C05463=1086.064,-73.363,-52.991,174.293,17.669,152.886
C05464=1086.058,-73.613,-52.980,174.292,17.667,152.886
C05465=1086.052,-73.862,-52.969,174.290,17.666,152.886
C05466=1086.046,-74.112,-52.958,174.289,17.665,152.886
C05467=1086.040,-74.362,-52.947,174.287,17.664,152.887
C05468=1086.034,-74.611,-52.936,174.286,17.662,152.886
C05469=1086.028,-74.861,-52.925,174.284,17.661,152.887
C05470=1086.021,-75.111,-52.914,174.282,17.660,152.887
C05471=1086.016,-75.360,-52.903,174.281,17.658,152.887
C05472=1086.010,-75.610,-52.892,174.279,17.657,152.887
C05473=1086.004,-75.860,-52.881,174.278,17.656,152.887
C05474=1085.998,-76.110,-52.870,174.277,17.655,152.887
C05475=1085.992,-76.359,-52.859,174.275,17.654,152.887
C05476=1085.986,-76.608,-52.849,174.274,17.653,152.887
C05477=1085.979,-76.858,-52.838,174.272,17.652,152.887
C05478=1085.974,-77.108,-52.827,174.271,17.650,152.887
C05479=1085.968,-77.358,-52.817,174.269,17.649,152.887
C05480=1085.962,-77.607,-52.806,174.268,17.648,152.887
C05481=1085.956,-77.858,-52.795,174.266,17.646,152.887
C05482=1085.950,-78.107,-52.785,174.265,17.645,152.887
C05483=1085.944,-78.356,-52.774,174.263,17.644,152.887
C05484=1085.938,-78.607,-52.762,174.261,17.643,152.887
C05485=1085.932,-78.856,-52.752,174.260,17.642,152.887
C05486=1085.926,-79.105,-52.741,174.258,17.640,152.887
C05487=1085.921,-79.356,-52.730,174.257,17.639,152.887
C05488=1085.914,-79.605,-52.720,174.255,17.638,152.888
C05489=1085.908,-79.855,-52.709,174.254,17.636,152.888
C05490=1085.902,-80.104,-52.698,174.252,17.635,152.888
C05491=1085.896,-80.354,-52.687,174.250,17.634,152.888
C05492=1085.889,-80.604,-52.677,174.250,17.634,152.888
C05493=1085.883,-80.879,-52.665,174.247,17.631,152.888
C05494=1085.876,-81.154,-52.654,174.246,17.630,152.888
C05495=1085.870,-81.429,-52.642,174.244,17.629,152.888
C05496=1085.863,-81.705,-52.629,174.243,17.628,152.888
C05497=1085.857,-81.955,-52.619,174.241,17.627,152.888
C05498=1085.851,-82.204,-52.609,174.239,17.626,152.888
C05499=1085.845,-82.454,-52.598,174.238,17.625,152.888
C05500=1085.839,-82.704,-52.587,174.236,17.623,152.888
C05501=1085.832,-82.953,-52.577,174.235,17.622,152.888
C05502=1085.827,-83.203,-52.566,174.233,17.621,152.889
C05503=1085.820,-83.452,-52.556,174.232,17.620,152.889
C05504=1085.814,-83.703,-52.545,174.231,17.619,152.889
C05505=1085.808,-83.952,-52.534,174.229,17.618,152.889
C05506=1085.802,-84.202,-52.524,174.227,17.617,152.889
C05507=1085.796,-84.451,-52.514,174.226,17.616,152.889
C05508=1085.790,-84.702,-52.502,174.224,17.615,152.889
C05509=1085.784,-84.951,-52.493,174.223,17.613,152.889
C05510=1085.778,-85.201,-52.482,174.221,17.612,152.889
C05511=1085.771,-85.450,-52.472,174.219,17.611,152.889
C05512=1085.766,-85.699,-52.461,174.218,17.610,152.889
C05513=1085.760,-85.950,-52.450,174.216,17.608,152.889
C05514=1085.753,-86.199,-52.440,174.216,17.608,152.889
C05515=1085.747,-86.449,-52.429,174.214,17.607,152.889
C05516=1085.741,-86.699,-52.419,174.212,17.606,152.890
C05517=1085.736,-86.948,-52.409,174.211,17.604,152.890
C05518=1085.729,-87.198,-52.397,174.209,17.603,152.890
C05519=1085.723,-87.448,-52.388,174.208,17.602,152.890
C05520=1085.717,-87.698,-52.377,174.206,17.601,152.890
C05521=1085.711,-87.947,-52.367,174.204,17.600,152.890
C05522=1085.705,-88.197,-52.356,174.203,17.599,152.890
C05523=1085.699,-88.446,-52.346,174.201,17.597,152.890
C05524=1085.693,-88.697,-52.336,174.200,17.596,152.890
C05525=1085.687,-88.947,-52.325,174.199,17.595,152.890
C05526=1085.681,-89.196,-52.314,174.197,17.594,152.890
C05527=1085.675,-89.446,-52.304,174.195,17.593,152.890
C05528=1085.669,-89.695,-52.294,174.194,17.592,152.891
C05529=1085.663,-89.945,-52.284,174.192,17.591,152.891
C05530=1085.656,-90.195,-52.273,174.191,17.590,152.891
C05531=1085.650,-90.444,-52.262,174.189,17.589,152.891
C05532=1085.645,-90.695,-52.252,174.187,17.587,152.891
C05533=1085.639,-90.944,-52.242,174.187,17.587,152.891
C05534=1085.633,-91.194,-52.232,174.185,17.586,152.891
C05535=1085.627,-91.443,-52.221,174.183,17.585,152.891
C05536=1085.621,-91.693,-52.211,174.182,17.583,152.891
C05537=1085.615,-91.942,-52.201,174.180,17.582,152.891
C05538=1085.609,-92.193,-52.190,174.179,17.581,152.891
C05539=1085.602,-92.442,-52.180,174.177,17.580,152.891
C05540=1085.597,-92.692,-52.170,174.175,17.579,152.892
C05541=1085.590,-92.942,-52.160,174.174,17.578,152.892
C05542=1085.585,-93.192,-52.150,174.173,17.577,152.892
C05543=1085.578,-93.441,-52.139,174.171,17.576,152.892
C05544=1085.573,-93.691,-52.129,174.170,17.575,152.892
C05545=1085.567,-93.940,-52.119,174.168,17.574,152.892
C05546=1085.561,-94.190,-52.109,174.166,17.573,152.892
C05547=1085.555,-94.439,-52.098,174.165,17.572,152.892
C05548=1085.549,-94.690,-52.088,174.163,17.570,152.892
C05549=1085.543,-94.939,-52.078,174.162,17.570,152.892
C05550=1085.537,-95.189,-52.068,174.161,17.569,152.892
C05551=1085.530,-95.439,-52.057,174.159,17.568,152.893
C05552=1085.525,-95.689,-52.047,174.157,17.567,152.893
C05553=1085.518,-95.938,-52.037,174.156,17.566,152.893
C05554=1085.513,-96.188,-52.027,174.154,17.564,152.893
C05555=1085.507,-96.438,-52.017,174.153,17.563,152.893
C05556=1085.501,-96.687,-52.006,174.152,17.563,152.893
C05557=1085.494,-96.964,-51.995,174.150,17.561,152.893
C05558=1085.488,-97.242,-51.984,174.148,17.560,152.893
C05559=1085.481,-97.520,-51.972,174.146,17.559,152.893
C05560=1085.474,-97.797,-51.962,174.144,17.558,152.893
C05561=1085.469,-98.047,-51.951,174.144,17.557,152.894
C05562=1085.462,-98.297,-51.941,174.142,17.556,152.894
C05563=1085.455,-98.547,-51.931,174.140,17.555,152.894
C05564=1085.450,-98.797,-51.921,174.139,17.554,152.894
C05565=1085.444,-99.046,-51.911,174.137,17.553,152.894
C05566=1085.437,-99.296,-51.901,174.135,17.552,152.894
C05567=1085.432,-99.546,-51.891,174.134,17.551,152.894
C05568=1085.425,-99.795,-51.881,174.133,17.550,152.894
C05569=1085.419,-100.045,-51.871,174.131,17.549,152.894
C05570=1085.414,-100.295,-51.861,174.129,17.548,152.894
C05571=1085.407,-100.544,-51.851,174.128,17.547,152.895
C05572=1085.401,-100.794,-51.841,174.126,17.546,152.895
C05573=1085.395,-101.044,-51.832,174.125,17.546,152.895
C05574=1085.389,-101.293,-51.821,174.123,17.545,152.895
C05575=1085.383,-101.543,-51.811,174.122,17.544,152.895
C05576=1085.377,-101.793,-51.802,174.120,17.543,152.895
C05577=1085.371,-102.043,-51.792,174.118,17.542,152.895
C05578=1085.365,-102.292,-51.781,174.117,17.541,152.895
C05579=1085.359,-102.542,-51.772,174.116,17.540,152.896
C05580=1085.353,-102.792,-51.762,174.114,17.539,152.896
C05581=1085.347,-103.041,-51.751,174.113,17.538,152.896
C05582=1085.341,-103.291,-51.742,174.111,17.537,152.896
C05583=1085.335,-103.541,-51.732,174.109,17.536,152.896
C05584=1085.328,-103.791,-51.722,174.108,17.535,152.896
C05585=1085.323,-104.041,-51.712,174.107,17.535,152.896
C05586=1085.317,-104.290,-51.702,174.105,17.534,152.896
C05587=1085.310,-104.540,-51.692,174.103,17.533,152.897
C05588=1085.304,-104.789,-51.683,174.102,17.532,152.897
C05589=1085.298,-105.039,-51.673,174.100,17.531,152.897
C05590=1085.292,-105.289,-51.662,174.099,17.530,152.897
C05591=1085.286,-105.538,-51.653,174.097,17.529,152.897
C05592=1085.280,-105.788,-51.643,174.096,17.528,152.897
C05593=1085.274,-106.038,-51.634,174.094,17.527,152.897
C05594=1085.268,-106.288,-51.624,174.092,17.526,152.897
C05595=1085.262,-106.537,-51.613,174.091,17.526,152.898
C05596=1085.256,-106.787,-51.604,174.090,17.525,152.898
C05597=1085.250,-107.037,-51.594,174.088,17.524,152.898
C05598=1085.243,-107.287,-51.585,174.086,17.523,152.898
C05599=1085.237,-107.537,-51.575,174.084,17.522,152.898
C05600=1085.232,-107.787,-51.565,174.084,17.522,152.898
C05601=1085.226,-108.036,-51.555,174.082,17.521,152.898
C05602=1085.219,-108.286,-51.545,174.080,17.519,152.898
C05603=1085.213,-108.535,-51.535,174.079,17.518,152.899
C05604=1085.207,-108.785,-51.526,174.078,17.518,152.899
C05605=1085.201,-109.035,-51.516,174.076,17.517,152.899
C05606=1085.194,-109.285,-51.507,174.074,17.516,152.899
C05607=1085.188,-109.535,-51.497,174.073,17.515,152.899
C05608=1085.182,-109.784,-51.488,174.071,17.515,152.899
C05609=1085.176,-110.034,-51.478,174.070,17.514,152.899
C05610=1085.169,-110.283,-51.468,174.068,17.513,152.900
C05611=1085.164,-110.534,-51.458,174.067,17.512,152.900
C05612=1085.158,-110.783,-51.448,174.065,17.511,152.900
C05613=1085.152,-111.033,-51.438,174.064,17.511,152.900
C05614=1085.145,-111.283,-51.429,174.062,17.510,152.900
C05615=1085.139,-111.533,-51.419,174.060,17.509,152.900
C05616=1085.133,-111.783,-51.410,174.059,17.508,152.900
C05617=1085.128,-112.032,-51.400,174.057,17.507,152.901
C05618=1085.121,-112.281,-51.391,174.056,17.507,152.901
C05619=1085.115,-112.531,-51.381,174.054,17.506,152.901
C05620=1085.109,-112.781,-51.372,174.052,17.505,152.901
C05621=1085.103,-113.054,-51.361,174.051,17.504,152.901
C05622=1085.095,-113.327,-51.350,174.049,17.503,152.901
C05623=1085.089,-113.600,-51.340,174.047,17.502,152.902
C05624=1085.082,-113.873,-51.330,174.046,17.501,152.902
C05625=1085.076,-114.123,-51.320,174.045,17.501,152.902
C05626=1085.070,-114.373,-51.311,174.043,17.500,152.902
C05627=1085.064,-114.622,-51.301,174.041,17.499,152.902
C05628=1085.058,-114.872,-51.292,174.040,17.498,152.902
C05629=1085.052,-115.122,-51.282,174.038,17.498,152.902
C05630=1085.046,-115.371,-51.273,174.037,17.497,152.903
C05631=1085.040,-115.621,-51.263,174.035,17.497,152.903
C05632=1085.033,-115.871,-51.254,174.033,17.495,152.903
C05633=1085.027,-116.121,-51.244,174.032,17.495,152.903
C05634=1085.021,-116.371,-51.234,174.030,17.494,152.903
C05635=1085.015,-116.620,-51.225,174.029,17.493,152.903
C05636=1085.009,-116.870,-51.215,174.027,17.492,152.903
C05637=1085.003,-117.120,-51.207,174.026,17.492,152.904
C05638=1084.997,-117.370,-51.197,174.024,17.491,152.904
C05639=1084.990,-117.619,-51.188,174.022,17.491,152.904
C05640=1084.984,-117.869,-51.179,174.022,17.490,152.904
C05641=1084.978,-118.119,-51.169,174.020,17.489,152.904
C05642=1084.972,-118.369,-51.160,174.018,17.489,152.905
C05643=1084.966,-118.618,-51.150,174.016,17.487,152.905
C05644=1084.959,-118.868,-51.140,174.015,17.487,152.905
C05645=1084.954,-119.117,-51.131,174.014,17.486,152.905
C05646=1084.948,-119.367,-51.122,174.012,17.486,152.905
C05647=1084.942,-119.617,-51.113,174.010,17.485,152.905
C05648=1084.936,-119.867,-51.103,174.009,17.484,152.905
C05649=1084.929,-120.117,-51.094,174.007,17.484,152.906
C05650=1084.923,-120.367,-51.085,174.006,17.483,152.906
C05651=1084.916,-120.616,-51.075,174.004,17.483,152.906
C05652=1084.911,-120.865,-51.066,174.003,17.482,152.906
C05653=1084.905,-121.116,-51.057,174.001,17.481,152.906
C05654=1084.899,-121.366,-51.048,173.999,17.480,152.906
C05655=1084.893,-121.615,-51.038,173.998,17.480,152.907
C05656=1084.886,-121.865,-51.029,173.996,17.479,152.907
C05657=1084.880,-122.115,-51.019,173.995,17.478,152.907
C05658=1084.874,-122.364,-51.010,173.994,17.478,152.907
C05659=1084.868,-122.614,-51.001,173.992,17.477,152.907
C05660=1084.862,-122.864,-50.992,173.990,17.476,152.908
C05661=1084.856,-123.114,-50.982,173.988,17.476,152.908
C05662=1084.849,-123.363,-50.973,173.987,17.475,152.908
C05663=1084.843,-123.614,-50.964,173.985,17.475,152.908
C05664=1084.837,-123.863,-50.955,173.984,17.474,152.908
C05665=1084.831,-124.113,-50.946,173.983,17.474,152.908
C05666=1084.825,-124.362,-50.936,173.981,17.472,152.909
C05667=1084.819,-124.613,-50.927,173.979,17.472,152.909
C05668=1084.812,-124.862,-50.918,173.978,17.471,152.909
C05669=1084.807,-125.111,-50.909,173.976,17.471,152.909
C05670=1084.801,-125.361,-50.899,173.975,17.470,152.909
C05671=1084.794,-125.611,-50.891,173.973,17.469,152.910
C05672=1084.788,-125.861,-50.882,173.972,17.469,152.910
C05673=1084.782,-126.111,-50.872,173.970,17.468,152.910
C05674=1084.775,-126.361,-50.863,173.968,17.468,152.910
C05675=1084.769,-126.610,-50.855,173.967,17.467,152.910
C05676=1084.763,-126.860,-50.845,173.965,17.467,152.910
C05677=1084.757,-127.110,-50.835,173.963,17.466,152.911
C05678=1084.750,-127.360,-50.827,173.963,17.466,152.911
C05679=1084.744,-127.610,-50.818,173.961,17.465,152.911
C05680=1084.739,-127.859,-50.808,173.959,17.464,152.911
C05681=1084.733,-128.116,-50.799,173.958,17.464,152.911
C05682=1084.731,-128.373,-50.789,173.957,17.462,152.911
C05683=1084.733,-128.628,-50.776,173.956,17.459,152.911
C05684=1084.740,-128.881,-50.763,173.955,17.454,152.910
C05685=1084.338,-128.903,-50.895,173.912,17.569,152.940
C05686=1084.332,-128.650,-50.909,173.912,17.573,152.941
C05687=1084.328,-128.394,-50.921,173.912,17.577,152.941
C05688=1084.331,-128.138,-50.932,173.914,17.578,152.941
C05689=1084.335,-127.881,-50.941,173.915,17.579,152.941
C05690=1084.342,-127.632,-50.950,173.917,17.580,152.941
C05691=1084.348,-127.382,-50.960,173.918,17.580,152.941
C05692=1084.354,-127.132,-50.969,173.920,17.581,152.941
C05693=1084.361,-126.882,-50.978,173.922,17.582,152.941
C05694=1084.367,-126.633,-50.987,173.923,17.582,152.940
C05695=1084.373,-126.383,-50.996,173.925,17.583,152.940
C05696=1084.379,-126.133,-51.005,173.927,17.584,152.940
C05697=1084.386,-125.883,-51.014,173.928,17.584,152.940
C05698=1084.392,-125.633,-51.023,173.929,17.585,152.940
C05699=1084.397,-125.384,-51.032,173.931,17.585,152.939
C05700=1084.404,-125.134,-51.041,173.933,17.586,152.939
C05701=1084.410,-124.884,-51.051,173.934,17.586,152.939
C05702=1084.416,-124.634,-51.060,173.936,17.587,152.939
C05703=1084.422,-124.384,-51.069,173.938,17.588,152.939
C05704=1084.428,-124.135,-51.078,173.938,17.588,152.939
C05705=1084.435,-123.886,-51.087,173.940,17.589,152.938
C05706=1084.441,-123.635,-51.096,173.942,17.590,152.938
C05707=1084.447,-123.385,-51.106,173.944,17.590,152.938
C05708=1084.453,-123.136,-51.115,173.945,17.591,152.938
C05709=1084.459,-122.886,-51.125,173.947,17.592,152.938
C05710=1084.466,-122.637,-51.133,173.948,17.593,152.937
C05711=1084.471,-122.387,-51.142,173.949,17.593,152.937
C05712=1084.478,-122.137,-51.152,173.951,17.594,152.937
C05713=1084.484,-121.887,-51.161,173.953,17.594,152.937
C05714=1084.490,-121.637,-51.171,173.955,17.595,152.937
C05715=1084.496,-121.387,-51.181,173.956,17.595,152.937
C05716=1084.501,-121.138,-51.189,173.957,17.596,152.936
C05717=1084.508,-120.888,-51.198,173.959,17.597,152.936
C05718=1084.514,-120.638,-51.208,173.961,17.598,152.936
C05719=1084.521,-120.389,-51.217,173.962,17.598,152.936
C05720=1084.527,-120.139,-51.227,173.964,17.599,152.936
C05721=1084.533,-119.889,-51.236,173.965,17.600,152.936
C05722=1084.538,-119.639,-51.245,173.966,17.601,152.936
C05723=1084.544,-119.390,-51.254,173.968,17.601,152.935
C05724=1084.551,-119.140,-51.264,173.970,17.602,152.935
C05725=1084.557,-118.890,-51.273,173.972,17.603,152.935
C05726=1084.564,-118.640,-51.282,173.973,17.603,152.935
C05727=1084.570,-118.391,-51.292,173.975,17.604,152.935
C05728=1084.576,-118.141,-51.302,173.976,17.605,152.934
C05729=1084.582,-117.891,-51.311,173.978,17.606,152.934
C05730=1084.588,-117.642,-51.320,173.979,17.606,152.934
C05731=1084.594,-117.392,-51.329,173.981,17.607,152.934
C05732=1084.600,-117.142,-51.339,173.982,17.608,152.934
C05733=1084.606,-116.892,-51.348,173.984,17.608,152.934
C05734=1084.612,-116.642,-51.358,173.985,17.609,152.934
C05735=1084.618,-116.392,-51.368,173.987,17.610,152.933
C05736=1084.624,-116.143,-51.377,173.989,17.611,152.933
C05737=1084.631,-115.893,-51.387,173.990,17.612,152.933
C05738=1084.638,-115.643,-51.396,173.991,17.612,152.933
C05739=1084.643,-115.394,-51.405,173.993,17.613,152.933
C05740=1084.649,-115.144,-51.414,173.995,17.614,152.933
C05741=1084.655,-114.895,-51.424,173.996,17.615,152.932
C05742=1084.662,-114.645,-51.434,173.998,17.615,152.932
C05743=1084.668,-114.395,-51.443,173.999,17.616,152.932
C05744=1084.674,-114.145,-51.453,174.001,17.617,152.932
C05745=1084.680,-113.895,-51.462,174.003,17.617,152.932
C05746=1084.686,-113.622,-51.473,174.004,17.619,152.932
C05747=1084.693,-113.348,-51.484,174.005,17.619,152.932
C05748=1084.700,-113.075,-51.494,174.007,17.620,152.931
C05749=1084.706,-112.802,-51.504,174.009,17.621,152.931
C05750=1084.712,-112.552,-51.514,174.011,17.622,152.931
C05751=1084.718,-112.303,-51.523,174.012,17.623,152.931
C05752=1084.725,-112.053,-51.533,174.014,17.624,152.931
C05753=1084.731,-111.803,-51.542,174.015,17.624,152.931
C05754=1084.737,-111.553,-51.552,174.017,17.625,152.931
C05755=1084.743,-111.303,-51.562,174.018,17.626,152.930
C05756=1084.749,-111.054,-51.571,174.020,17.627,152.930
C05757=1084.755,-110.804,-51.581,174.022,17.628,152.930
C05758=1084.762,-110.555,-51.591,174.023,17.628,152.930
C05759=1084.768,-110.305,-51.601,174.024,17.629,152.930
C05760=1084.774,-110.055,-51.610,174.026,17.630,152.930
C05761=1084.780,-109.805,-51.620,174.028,17.631,152.929
C05762=1084.786,-109.555,-51.630,174.029,17.631,152.929
C05763=1084.791,-109.306,-51.639,174.030,17.632,152.929
C05764=1084.798,-109.056,-51.649,174.032,17.633,152.929
C05765=1084.804,-108.806,-51.658,174.034,17.634,152.929
C05766=1084.810,-108.557,-51.668,174.036,17.635,152.929
C05767=1084.816,-108.307,-51.678,174.036,17.635,152.929
C05768=1084.823,-108.058,-51.688,174.038,17.637,152.929
C05769=1084.829,-107.808,-51.697,174.040,17.638,152.929
C05770=1084.835,-107.558,-51.707,174.041,17.639,152.928
C05771=1084.840,-107.308,-51.717,174.043,17.640,152.928
C05772=1084.846,-107.058,-51.726,174.044,17.640,152.928
C05773=1084.853,-106.808,-51.736,174.046,17.641,152.928
C05774=1084.859,-106.559,-51.746,174.048,17.642,152.928
C05775=1084.865,-106.309,-51.756,174.049,17.643,152.928
C05776=1084.871,-106.060,-51.765,174.051,17.644,152.928
C05777=1084.877,-105.809,-51.776,174.052,17.644,152.928
C05778=1084.883,-105.560,-51.785,174.053,17.646,152.927
C05779=1084.890,-105.311,-51.795,174.055,17.647,152.927
C05780=1084.896,-105.061,-51.805,174.057,17.648,152.927
C05781=1084.901,-104.811,-51.815,174.059,17.648,152.927
C05782=1084.907,-104.561,-51.825,174.059,17.649,152.927
C05783=1084.913,-104.311,-51.834,174.061,17.650,152.927
C05784=1084.920,-104.062,-51.845,174.063,17.651,152.927
C05785=1084.925,-103.812,-51.855,174.064,17.652,152.927
C05786=1084.932,-103.562,-51.864,174.066,17.653,152.926
C05787=1084.938,-103.312,-51.874,174.068,17.654,152.926
C05788=1084.944,-103.063,-51.884,174.069,17.654,152.926
C05789=1084.950,-102.813,-51.894,174.070,17.656,152.926
C05790=1084.956,-102.563,-51.904,174.072,17.657,152.926
C05791=1084.962,-102.313,-51.913,174.074,17.658,152.926
C05792=1084.968,-102.064,-51.924,174.075,17.659,152.926
C05793=1084.974,-101.814,-51.934,174.076,17.659,152.926
C05794=1084.980,-101.564,-51.944,174.078,17.660,152.926
C05795=1084.987,-101.315,-51.954,174.079,17.661,152.926
C05796=1084.993,-101.065,-51.963,174.081,17.662,152.925
C05797=1084.998,-100.815,-51.974,174.083,17.663,152.925
C05798=1085.005,-100.566,-51.984,174.084,17.665,152.925
C05799=1085.011,-100.316,-51.993,174.085,17.665,152.925
C05800=1085.016,-100.066,-52.004,174.087,17.666,152.925
C05801=1085.023,-99.816,-52.014,174.088,17.667,152.925
C05802=1085.030,-99.566,-52.024,174.090,17.668,152.925
C05803=1085.036,-99.316,-52.033,174.092,17.669,152.925
C05804=1085.041,-99.067,-52.044,174.093,17.670,152.925
C05805=1085.048,-98.817,-52.054,174.095,17.671,152.924
C05806=1085.054,-98.567,-52.063,174.096,17.672,152.924
C05807=1085.059,-98.318,-52.074,174.098,17.673,152.924
C05808=1085.066,-98.068,-52.084,174.099,17.674,152.924
C05809=1085.072,-97.818,-52.093,174.101,17.675,152.924
C05810=1085.078,-97.540,-52.105,174.103,17.676,152.924
C05811=1085.085,-97.263,-52.116,174.104,17.677,152.924
C05812=1085.091,-96.986,-52.128,174.106,17.678,152.924
C05813=1085.098,-96.708,-52.139,174.108,17.679,152.924
C05814=1085.104,-96.458,-52.149,174.109,17.680,152.923
C05815=1085.110,-96.209,-52.159,174.111,17.681,152.923
C05816=1085.116,-95.959,-52.169,174.113,17.682,152.923
C05817=1085.122,-95.709,-52.180,174.114,17.684,152.923
C05818=1085.128,-95.459,-52.190,174.115,17.685,152.923
C05819=1085.134,-95.210,-52.200,174.116,17.686,152.923
C05820=1085.140,-94.959,-52.211,174.118,17.687,152.923
C05821=1085.146,-94.709,-52.220,174.120,17.688,152.923
C05822=1085.152,-94.460,-52.231,174.121,17.689,152.923
C05823=1085.158,-94.210,-52.241,174.123,17.690,152.923
C05824=1085.164,-93.961,-52.252,174.124,17.691,152.923
C05825=1085.170,-93.711,-52.261,174.126,17.693,152.923
C05826=1085.176,-93.461,-52.272,174.127,17.693,152.922
C05827=1085.182,-93.212,-52.282,174.129,17.694,152.922
C05828=1085.188,-92.962,-52.292,174.130,17.695,152.922
C05829=1085.194,-92.712,-52.302,174.132,17.696,152.922
C05830=1085.200,-92.463,-52.313,174.134,17.697,152.922
C05831=1085.206,-92.213,-52.323,174.135,17.699,152.922
C05832=1085.212,-91.963,-52.334,174.137,17.700,152.922
C05833=1085.218,-91.713,-52.343,174.138,17.701,152.922
C05834=1085.224,-91.464,-52.354,174.139,17.701,152.922
C05835=1085.231,-91.214,-52.364,174.141,17.703,152.922
C05836=1085.236,-90.964,-52.375,174.142,17.704,152.922
C05837=1085.243,-90.715,-52.385,174.144,17.705,152.922
C05838=1085.248,-90.465,-52.395,174.145,17.706,152.921
C05839=1085.254,-90.215,-52.406,174.147,17.707,152.921
C05840=1085.261,-89.965,-52.416,174.149,17.708,152.921
C05841=1085.266,-89.715,-52.427,174.150,17.710,152.921
C05842=1085.273,-89.466,-52.437,174.152,17.711,152.921
C05843=1085.278,-89.216,-52.447,174.153,17.712,152.921
C05844=1085.285,-88.967,-52.458,174.154,17.713,152.921
C05845=1085.290,-88.717,-52.468,174.156,17.714,152.921
C05846=1085.296,-88.467,-52.479,174.157,17.715,152.921
C05847=1085.303,-88.218,-52.489,174.159,17.716,152.921
C05848=1085.308,-87.967,-52.499,174.161,17.717,152.921
C05849=1085.315,-87.718,-52.510,174.162,17.718,152.921
C05850=1085.321,-87.469,-52.521,174.164,17.720,152.921
C05851=1085.327,-87.219,-52.530,174.165,17.721,152.921
C05852=1085.333,-86.969,-52.541,174.167,17.722,152.920
C05853=1085.339,-86.719,-52.552,174.168,17.723,152.920
C05854=1085.345,-86.469,-52.562,174.170,17.724,152.920
C05855=1085.351,-86.220,-52.573,174.171,17.725,152.920
C05856=1085.357,-85.971,-52.583,174.173,17.726,152.920
C05857=1085.363,-85.720,-52.593,174.174,17.727,152.920
C05858=1085.369,-85.470,-52.604,174.176,17.729,152.920
C05859=1085.375,-85.221,-52.615,174.177,17.730,152.920
C05860=1085.381,-84.971,-52.625,174.179,17.731,152.920
C05861=1085.387,-84.722,-52.635,174.181,17.732,152.920
C05862=1085.394,-84.472,-52.646,174.182,17.734,152.920
C05863=1085.399,-84.222,-52.657,174.184,17.735,152.920
C05864=1085.406,-83.973,-52.667,174.185,17.736,152.920
C05865=1085.411,-83.723,-52.678,174.186,17.736,152.919
C05866=1085.418,-83.473,-52.689,174.188,17.738,152.920
C05867=1085.424,-83.224,-52.699,174.189,17.739,152.919
C05868=1085.430,-82.974,-52.709,174.191,17.740,152.919
C05869=1085.436,-82.724,-52.720,174.192,17.742,152.919
C05870=1085.442,-82.474,-52.731,174.194,17.743,152.919
C05871=1085.448,-82.225,-52.742,174.196,17.744,152.919
C05872=1085.454,-81.975,-52.751,174.197,17.745,152.919
C05873=1085.460,-81.725,-52.762,174.199,17.746,152.919
C05874=1085.467,-81.450,-52.774,174.200,17.747,152.919
C05875=1085.474,-81.175,-52.786,174.202,17.748,152.919
C05876=1085.480,-80.899,-52.797,174.203,17.750,152.919
C05877=1085.487,-80.624,-52.810,174.205,17.751,152.919
C05878=1085.493,-80.374,-52.821,174.207,17.752,152.919
C05879=1085.500,-80.125,-52.831,174.208,17.754,152.919
C05880=1085.506,-79.874,-52.841,174.210,17.755,152.919
C05881=1085.511,-79.625,-52.852,174.211,17.756,152.918
C05882=1085.517,-79.375,-52.863,174.213,17.757,152.918
C05883=1085.524,-79.126,-52.873,174.214,17.758,152.918
C05884=1085.530,-78.876,-52.885,174.216,17.760,152.918
C05885=1085.536,-78.626,-52.896,174.218,17.761,152.918
C05886=1085.541,-78.377,-52.906,174.219,17.762,152.918
C05887=1085.547,-78.127,-52.917,174.221,17.764,152.918
C05888=1085.553,-77.876,-52.928,174.222,17.765,152.918
C05889=1085.560,-77.627,-52.938,174.224,17.766,152.918
C05890=1085.565,-77.378,-52.949,174.225,17.767,152.918
C05891=1085.572,-77.128,-52.960,174.227,17.769,152.918
C05892=1085.577,-76.878,-52.971,174.228,17.770,152.918
C05893=1085.583,-76.629,-52.982,174.230,17.771,152.918
C05894=1085.589,-76.379,-52.993,174.231,17.773,152.918
C05895=1085.596,-76.129,-53.003,174.232,17.773,152.918
C05896=1085.602,-75.880,-53.014,174.234,17.775,152.918
C05897=1085.608,-75.630,-53.025,174.235,17.776,152.918
C05898=1085.614,-75.380,-53.036,174.237,17.777,152.918
C05899=1085.620,-75.131,-53.047,174.238,17.778,152.918
C05900=1085.625,-74.881,-53.058,174.240,17.780,152.918
C05901=1085.631,-74.632,-53.069,174.241,17.781,152.918
C05902=1085.637,-74.381,-53.080,174.243,17.782,152.917
C05903=1085.644,-74.132,-53.091,174.244,17.784,152.918
C05904=1085.649,-73.882,-53.101,174.246,17.785,152.917
C05905=1085.656,-73.632,-53.112,174.247,17.786,152.917
C05906=1085.661,-73.382,-53.124,174.249,17.788,152.918
C05907=1085.666,-73.133,-53.134,174.251,17.789,152.917
C05908=1085.672,-72.884,-53.146,174.252,17.791,152.917
C05909=1085.679,-72.634,-53.157,174.254,17.792,152.917
C05910=1085.685,-72.384,-53.168,174.255,17.793,152.917
C05911=1085.690,-72.135,-53.179,174.257,17.794,152.917
C05912=1085.697,-71.884,-53.190,174.258,17.796,152.917
C05913=1085.702,-71.635,-53.201,174.259,17.797,152.917
C05914=1085.708,-71.385,-53.212,174.261,17.798,152.917
C05915=1085.714,-71.136,-53.223,174.262,17.800,152.917
C05916=1085.720,-70.886,-53.234,174.264,17.801,152.917
C05917=1085.726,-70.636,-53.245,174.266,17.803,152.917
C05918=1085.732,-70.387,-53.256,174.267,17.804,152.917
C05919=1085.738,-70.137,-53.267,174.269,17.805,152.917
C05920=1085.744,-69.887,-53.278,174.270,17.807,152.917
C05921=1085.749,-69.637,-53.289,174.272,17.808,152.917
C05922=1085.755,-69.387,-53.301,174.273,17.809,152.917
C05923=1085.761,-69.138,-53.312,174.275,17.811,152.917
C05924=1085.767,-68.889,-53.323,174.276,17.812,152.917
C05925=1085.773,-68.639,-53.334,174.277,17.814,152.917
C05926=1085.779,-68.389,-53.345,174.279,17.815,152.917
C05927=1085.785,-68.140,-53.356,174.281,17.816,152.917
C05928=1085.791,-67.889,-53.367,174.282,17.817,152.917
C05929=1085.797,-67.640,-53.378,174.284,17.819,152.917
C05930=1085.802,-67.390,-53.390,174.285,17.821,152.917
C05931=1085.808,-67.141,-53.402,174.287,17.822,152.917
C05932=1085.814,-66.891,-53.413,174.288,17.823,152.917
C05933=1085.820,-66.642,-53.423,174.290,17.824,152.917
C05934=1085.826,-66.391,-53.435,174.291,17.826,152.917
C05935=1085.832,-66.142,-53.446,174.292,17.827,152.917
C05936=1085.839,-65.892,-53.458,174.294,17.828,152.917
C05937=1085.844,-65.643,-53.468,174.296,17.830,152.917
C05938=1085.851,-65.369,-53.481,174.297,17.832,152.917
C05939=1085.857,-65.096,-53.494,174.299,17.833,152.917
C05940=1085.864,-64.823,-53.506,174.301,17.835,152.917
C05941=1085.869,-64.550,-53.518,174.302,17.836,152.917
C05942=1085.876,-64.300,-53.530,174.304,17.837,152.917
C05943=1085.882,-64.051,-53.541,174.305,17.839,152.917
C05944=1085.888,-63.800,-53.552,174.307,17.840,152.917
C05945=1085.894,-63.551,-53.563,174.308,17.842,152.917
C05946=1085.900,-63.302,-53.574,174.310,17.843,152.917
C05947=1085.905,-63.052,-53.586,174.311,17.845,152.917
C05948=1085.911,-62.802,-53.597,174.313,17.846,152.917
C05949=1085.917,-62.552,-53.608,174.314,17.847,152.917
C05950=1085.924,-62.303,-53.620,174.316,17.849,152.917
C05951=1085.930,-62.053,-53.631,174.317,17.850,152.917
C05952=1085.935,-61.803,-53.642,174.319,17.852,152.917
C05953=1085.941,-61.553,-53.654,174.320,17.853,152.916
C05954=1085.947,-61.304,-53.665,174.322,17.854,152.916
C05955=1085.953,-61.055,-53.676,174.323,17.856,152.917
C05956=1085.960,-60.805,-53.688,174.325,17.857,152.916
C05957=1085.965,-60.555,-53.700,174.326,17.858,152.916
C05958=1085.971,-60.305,-53.711,174.328,17.860,152.916
C05959=1085.977,-60.056,-53.722,174.329,17.861,152.916
C05960=1085.983,-59.806,-53.734,174.331,17.863,152.916
C05961=1085.989,-59.557,-53.745,174.333,17.865,152.916
C05962=1085.995,-59.307,-53.757,174.334,17.866,152.916
C05963=1086.001,-59.057,-53.768,174.336,17.867,152.916
C05964=1086.007,-58.807,-53.780,174.337,17.869,152.916
C05965=1086.013,-58.558,-53.791,174.339,17.870,152.916
C05966=1086.020,-58.308,-53.803,174.340,17.871,152.916
C05967=1086.025,-58.059,-53.814,174.342,17.873,152.916
C05968=1086.031,-57.808,-53.826,174.343,17.875,152.916
C05969=1086.037,-57.560,-53.837,174.345,17.876,152.916
C05970=1086.043,-57.309,-53.848,174.346,17.877,152.916
C05971=1086.049,-57.060,-53.861,174.348,17.879,152.916
C05972=1086.055,-56.810,-53.872,174.349,17.880,152.916
C05973=1086.061,-56.561,-53.883,174.351,17.881,152.916
C05974=1086.068,-56.311,-53.895,174.352,17.883,152.916
C05975=1086.073,-56.061,-53.907,174.354,17.884,152.916
C05976=1086.079,-55.812,-53.918,174.355,17.886,152.916
C05977=1086.086,-55.561,-53.929,174.356,17.887,152.916
C05978=1086.092,-55.312,-53.941,174.358,17.889,152.916
C05979=1086.097,-55.062,-53.953,174.360,17.890,152.916
C05980=1086.103,-54.813,-53.964,174.361,17.891,152.916
C05981=1086.110,-54.564,-53.976,174.362,17.893,152.916
C05982=1086.115,-54.313,-53.988,174.365,17.895,152.916
C05983=1086.121,-54.064,-54.000,174.366,17.896,152.916
C05984=1086.128,-53.814,-54.011,174.368,17.898,152.916
C05985=1086.134,-53.565,-54.023,174.369,17.899,152.916
C05986=1086.139,-53.315,-54.034,174.371,17.900,152.916
C05987=1086.146,-53.066,-54.046,174.372,17.902,152.916
C05988=1086.152,-52.816,-54.057,174.373,17.903,152.916
C05989=1086.158,-52.566,-54.070,174.375,17.905,152.916
C05990=1086.164,-52.316,-54.081,174.377,17.906,152.916
C05991=1086.170,-52.067,-54.093,174.378,17.908,152.916
C05992=1086.176,-51.818,-54.104,174.379,17.909,152.916
C05993=1086.182,-51.567,-54.116,174.381,17.910,152.916
C05994=1086.188,-51.318,-54.128,174.382,17.912,152.916
C05995=1086.194,-51.068,-54.139,174.384,17.913,152.916
C05996=1086.200,-50.818,-54.151,174.385,17.915,152.916
C05997=1086.207,-50.569,-54.163,174.388,17.917,152.916
C05998=1086.212,-50.319,-54.174,174.389,17.918,152.916
C05999=1086.218,-50.069,-54.187,174.390,17.920,152.916
C06000=1086.224,-49.820,-54.199,174.392,17.921,152.916
C06001=1086.230,-49.570,-54.210,174.394,17.922,152.916
C06002=1086.236,-49.298,-54.224,174.395,17.924,152.916
C06003=1086.242,-49.026,-54.236,174.396,17.926,152.916
C06004=1086.249,-48.754,-54.249,174.399,17.928,152.916
C06005=1086.256,-48.483,-54.262,174.400,17.929,152.916
C06006=1086.261,-48.233,-54.274,174.401,17.931,152.916
C06007=1086.267,-47.984,-54.286,174.403,17.932,152.916
C06008=1086.273,-47.734,-54.298,174.404,17.934,152.916
C06009=1086.279,-47.483,-54.310,174.406,17.935,152.916
C06010=1086.285,-47.234,-54.322,174.407,17.937,152.916
C06011=1086.291,-46.985,-54.334,174.409,17.939,152.916
C06012=1086.297,-46.736,-54.346,174.411,17.940,152.916
C06013=1086.303,-46.485,-54.358,174.412,17.942,152.916
C06014=1086.308,-46.235,-54.370,174.414,17.943,152.916
C06015=1086.314,-45.986,-54.382,174.415,17.945,152.916
C06016=1086.320,-45.736,-54.393,174.416,17.946,152.916
C06017=1086.326,-45.487,-54.405,174.418,17.948,152.917
C06018=1086.332,-45.237,-54.418,174.419,17.950,152.917
C06019=1086.339,-44.988,-54.430,174.421,17.951,152.916
C06020=1086.344,-44.738,-54.442,174.422,17.952,152.916
C06021=1086.350,-44.488,-54.454,174.424,17.954,152.916
C06022=1086.356,-44.238,-54.466,174.426,17.956,152.917
C06023=1086.362,-43.989,-54.478,174.427,17.957,152.917
C06024=1086.367,-43.739,-54.490,174.429,17.959,152.917
C06025=1086.374,-43.490,-54.502,174.430,17.961,152.917
C06026=1086.379,-43.240,-54.514,174.431,17.962,152.917
C06027=1086.386,-42.990,-54.526,174.433,17.963,152.917
C06028=1086.392,-42.740,-54.538,174.435,17.965,152.917
C06029=1086.397,-42.491,-54.550,174.436,17.966,152.917
C06030=1086.404,-42.242,-54.562,174.438,17.968,152.917
C06031=1086.410,-41.992,-54.575,174.440,17.970,152.917
C06032=1086.415,-41.742,-54.586,174.441,17.972,152.917
C06033=1086.421,-41.492,-54.598,174.442,17.973,152.917
C06034=1086.427,-41.243,-54.611,174.444,17.975,152.917
C06035=1086.432,-40.993,-54.623,174.445,17.976,152.917
C06036=1086.439,-40.744,-54.635,174.447,17.977,152.917
C06037=1086.445,-40.494,-54.648,174.448,17.979,152.917
C06038=1086.452,-40.244,-54.660,174.450,17.981,152.917
C06039=1086.457,-39.995,-54.672,174.452,17.983,152.917
C06040=1086.463,-39.745,-54.684,174.453,17.984,152.917
C06041=1086.469,-39.496,-54.696,174.455,17.986,152.917
C06042=1086.474,-39.246,-54.708,174.456,17.987,152.917
C06043=1086.480,-38.996,-54.720,174.457,17.989,152.917
C06044=1086.487,-38.746,-54.732,174.459,17.990,152.917
C06045=1086.493,-38.497,-54.745,174.460,17.992,152.917
C06046=1086.498,-38.247,-54.757,174.463,17.994,152.917
C06047=1086.504,-37.997,-54.770,174.464,17.995,152.917
C06048=1086.510,-37.748,-54.782,174.466,17.997,152.917
C06049=1086.515,-37.498,-54.794,174.467,17.998,152.917
C06050=1086.522,-37.249,-54.806,174.468,18.000,152.917
C06051=1086.528,-36.999,-54.819,174.470,18.001,152.917
C06052=1086.533,-36.750,-54.831,174.471,18.003,152.917
C06053=1086.539,-36.500,-54.844,174.473,18.005,152.917
C06054=1086.545,-36.250,-54.856,174.475,18.007,152.917
C06055=1086.551,-36.000,-54.869,174.476,18.008,152.917
C06056=1086.557,-35.751,-54.880,174.478,18.010,152.917
C06057=1086.563,-35.501,-54.893,174.479,18.011,152.917
C06058=1086.569,-35.251,-54.905,174.480,18.013,152.917
C06059=1086.574,-35.002,-54.918,174.482,18.015,152.917
C06060=1086.580,-34.752,-54.930,174.484,18.017,152.917
C06061=1086.586,-34.503,-54.943,174.485,18.018,152.917
C06062=1086.592,-34.253,-54.955,174.487,18.020,152.917
C06063=1086.597,-34.004,-54.968,174.488,18.021,152.918
C06064=1086.604,-33.755,-54.980,174.490,18.023,152.918
C06065=1086.610,-33.505,-54.993,174.491,18.024,152.918
C06066=1086.616,-33.233,-55.006,174.493,18.027,152.918
C06067=1086.623,-32.961,-55.019,174.495,18.028,152.918
C06068=1086.629,-32.690,-55.034,174.496,18.030,152.918
C06069=1086.635,-32.418,-55.047,174.498,18.032,152.918
C06070=1086.641,-32.169,-55.060,174.500,18.033,152.918
C06071=1086.647,-31.919,-55.072,174.501,18.035,152.918
C06072=1086.653,-31.669,-55.084,174.502,18.036,152.918
C06073=1086.659,-31.420,-55.096,174.504,18.038,152.918
C06074=1086.665,-31.171,-55.110,174.505,18.040,152.918
C06075=1086.671,-30.921,-55.122,174.507,18.042,152.918
C06076=1086.677,-30.671,-55.135,174.509,18.043,152.918
C06077=1086.683,-30.421,-55.147,174.510,18.045,152.918
C06078=1086.688,-30.172,-55.160,174.512,18.046,152.918
C06079=1086.694,-29.922,-55.172,174.513,18.048,152.918
C06080=1086.700,-29.673,-55.185,174.514,18.050,152.918
C06081=1086.706,-29.423,-55.198,174.517,18.052,152.918
C06082=1086.712,-29.173,-55.210,174.518,18.053,152.918
C06083=1086.718,-28.923,-55.222,174.519,18.055,152.918
C06084=1086.724,-28.675,-55.235,174.521,18.056,152.918
C06085=1086.730,-28.425,-55.248,174.522,18.058,152.918
C06086=1086.736,-28.175,-55.260,174.524,18.059,152.918
C06087=1086.742,-27.925,-55.273,174.526,18.062,152.918
C06088=1086.748,-27.676,-55.286,174.527,18.063,152.918
C06089=1086.754,-27.426,-55.299,174.529,18.065,152.918
C06090=1086.760,-27.176,-55.311,174.530,18.066,152.918
C06091=1086.766,-26.926,-55.324,174.532,18.068,152.918
C06092=1086.771,-26.678,-55.337,174.533,18.069,152.918
C06093=1086.777,-26.428,-55.349,174.535,18.071,152.918
C06094=1086.783,-26.178,-55.362,174.537,18.073,152.919
C06095=1086.789,-25.928,-55.376,174.538,18.075,152.919
C06096=1086.795,-25.678,-55.388,174.539,18.077,152.919
C06097=1086.800,-25.429,-55.401,174.541,18.078,152.919
C06098=1086.806,-25.179,-55.413,174.542,18.080,152.919
C06099=1086.812,-24.930,-55.426,174.544,18.082,152.919
C06100=1086.818,-24.680,-55.439,174.546,18.083,152.919
C06101=1086.824,-24.430,-55.451,174.547,18.085,152.919
C06102=1086.830,-24.181,-55.465,174.548,18.087,152.919
C06103=1086.835,-23.931,-55.478,174.550,18.088,152.919
C06104=1086.841,-23.682,-55.491,174.552,18.090,152.919
C06105=1086.847,-23.432,-55.503,174.553,18.092,152.919
C06106=1086.853,-23.182,-55.516,174.555,18.093,152.919
C06107=1086.859,-22.933,-55.529,174.556,18.095,152.919
C06108=1086.865,-22.683,-55.542,174.558,18.097,152.919
C06109=1086.870,-22.434,-55.556,174.560,18.099,152.919
C06110=1086.876,-22.184,-55.568,174.561,18.101,152.919
C06111=1086.882,-21.934,-55.581,174.562,18.102,152.919
C06112=1086.888,-21.685,-55.594,174.564,18.104,152.919
C06113=1086.894,-21.436,-55.606,174.565,18.105,152.919
C06114=1086.900,-21.186,-55.619,174.567,18.107,152.920
C06115=1086.905,-20.936,-55.633,174.569,18.109,152.920
C06116=1086.911,-20.687,-55.646,174.570,18.111,152.920
C06117=1086.917,-20.437,-55.658,174.572,18.112,152.920
C06118=1086.923,-20.187,-55.671,174.573,18.114,152.920
C06119=1086.929,-19.938,-55.684,174.574,18.115,152.920
C06120=1086.934,-19.688,-55.697,174.577,18.117,152.920
C06121=1086.941,-19.438,-55.711,174.578,18.119,152.920
C06122=1086.946,-19.188,-55.723,174.579,18.121,152.920
C06123=1086.953,-18.939,-55.736,174.581,18.123,152.920
C06124=1086.959,-18.689,-55.749,174.582,18.124,152.920
C06125=1086.964,-18.440,-55.763,174.584,18.126,152.920
C06126=1086.970,-18.191,-55.776,174.586,18.128,152.920
C06127=1086.976,-17.941,-55.788,174.587,18.129,152.920
C06128=1086.982,-17.692,-55.802,174.588,18.131,152.920
C06129=1086.988,-17.442,-55.814,174.591,18.133,152.920
C06130=1086.994,-17.169,-55.828,174.592,18.135,152.920
C06131=1087.000,-16.897,-55.843,174.593,18.136,152.920
C06132=1087.007,-16.625,-55.858,174.596,18.138,152.920
C06133=1087.013,-16.352,-55.871,174.597,18.140,152.920
C06134=1087.019,-16.103,-55.885,174.598,18.142,152.920
C06135=1087.025,-15.854,-55.898,174.601,18.144,152.920
C06136=1087.031,-15.604,-55.911,174.602,18.146,152.920
C06137=1087.037,-15.354,-55.924,174.603,18.147,152.921
C06138=1087.042,-15.104,-55.937,174.605,18.149,152.921
C06139=1087.049,-14.855,-55.951,174.606,18.150,152.921
C06140=1087.055,-14.606,-55.964,174.608,18.152,152.921
C06141=1087.060,-14.356,-55.977,174.610,18.154,152.921
C06142=1087.066,-14.106,-55.990,174.611,18.155,152.921
C06143=1087.072,-13.857,-56.004,174.612,18.158,152.921
C06144=1087.078,-13.607,-56.017,174.615,18.160,152.921
C06145=1087.083,-13.357,-56.031,174.616,18.161,152.921
C06146=1087.089,-13.108,-56.044,174.617,18.163,152.921
C06147=1087.095,-12.858,-56.056,174.619,18.164,152.921
C06148=1087.101,-12.608,-56.070,174.620,18.166,152.921
C06149=1087.107,-12.359,-56.084,174.622,18.168,152.921
C06150=1087.112,-12.109,-56.097,174.624,18.170,152.921
C06151=1087.118,-11.860,-56.110,174.625,18.172,152.921
C06152=1087.124,-11.610,-56.124,174.626,18.173,152.921
C06153=1087.130,-11.360,-56.136,174.629,18.175,152.921
C06154=1087.136,-11.111,-56.150,174.630,18.177,152.921
C06155=1087.141,-10.861,-56.164,174.631,18.178,152.921
C06156=1087.148,-10.612,-56.177,174.633,18.180,152.921
C06157=1087.153,-10.362,-56.190,174.635,18.182,152.921
C06158=1087.159,-10.113,-56.203,174.636,18.184,152.922
C06159=1087.164,-9.863,-56.217,174.638,18.186,152.922
C06160=1087.171,-9.614,-56.230,174.639,18.187,152.922
C06161=1087.176,-9.364,-56.244,174.640,18.189,152.922
C06162=1087.182,-9.114,-56.257,174.643,18.191,152.922
C06163=1087.188,-8.865,-56.271,174.644,18.192,152.922
C06164=1087.194,-8.616,-56.284,174.645,18.194,152.922
C06165=1087.199,-8.366,-56.298,174.647,18.196,152.922
C06166=1087.206,-8.116,-56.311,174.649,18.198,152.922
C06167=1087.212,-7.866,-56.324,174.650,18.199,152.922
C06168=1087.217,-7.617,-56.338,174.652,18.201,152.922
C06169=1087.224,-7.367,-56.351,174.653,18.203,152.922
C06170=1087.229,-7.118,-56.365,174.655,18.205,152.922
C06171=1087.235,-6.869,-56.378,174.657,18.207,152.922
C06172=1087.241,-6.619,-56.392,174.658,18.208,152.922
C06173=1087.247,-6.370,-56.405,174.659,18.210,152.922
C06174=1087.252,-6.119,-56.418,174.662,18.212,152.922
C06175=1087.258,-5.870,-56.432,174.663,18.213,152.922
C06176=1087.264,-5.621,-56.446,174.665,18.215,152.922
C06177=1087.270,-5.370,-56.460,174.666,18.217,152.923
C06178=1087.276,-5.121,-56.473,174.668,18.219,152.923
C06179=1087.282,-4.872,-56.487,174.669,18.221,152.923
C06180=1087.288,-4.622,-56.500,174.671,18.222,152.923
C06181=1087.293,-4.373,-56.514,174.672,18.224,152.923
C06182=1087.300,-4.123,-56.527,174.674,18.226,152.923
C06183=1087.305,-3.874,-56.541,174.676,18.227,152.923
C06184=1087.312,-3.624,-56.555,174.677,18.229,152.923
C06185=1087.317,-3.374,-56.569,174.679,18.230,152.923
C06186=1087.324,-3.125,-56.582,174.681,18.233,152.923
C06187=1087.329,-2.875,-56.596,174.682,18.235,152.923
C06188=1087.334,-2.626,-56.610,174.683,18.236,152.923
C06189=1087.340,-2.376,-56.624,174.685,18.238,152.923
C06190=1087.346,-2.127,-56.637,174.687,18.240,152.923
C06191=1087.352,-1.877,-56.651,174.688,18.241,152.923
C06192=1087.357,-1.628,-56.665,174.690,18.243,152.923
C06193=1087.363,-1.378,-56.678,174.691,18.245,152.923
C06194=1087.369,-1.103,-56.693,174.693,18.247,152.923
C06195=1087.376,-0.830,-56.708,174.695,18.249,152.923
C06196=1087.382,-0.556,-56.723,174.697,18.251,152.924
C06197=1087.388,-0.282,-56.739,174.698,18.253,152.924
C06198=1087.394,-0.032,-56.753,174.700,18.255,152.924
C06199=1087.399,0.217,-56.766,174.702,18.256,152.924
C06200=1087.405,0.467,-56.780,174.703,18.258,152.924
C06201=1087.411,0.716,-56.794,174.704,18.260,152.924
C06202=1087.417,0.966,-56.808,174.706,18.262,152.924
C06203=1087.423,1.216,-56.822,174.708,18.264,152.924
C06204=1087.428,1.466,-56.836,174.709,18.265,152.924
C06205=1087.434,1.715,-56.850,174.712,18.267,152.924
C06206=1087.440,1.964,-56.863,174.713,18.269,152.924
C06207=1087.446,2.213,-56.877,174.714,18.271,152.924
C06208=1087.451,2.463,-56.891,174.716,18.273,152.924
C06209=1087.457,2.713,-56.905,174.718,18.275,152.924
C06210=1087.463,2.963,-56.919,174.719,18.276,152.924
C06211=1087.469,3.212,-56.933,174.721,18.278,152.924
C06212=1087.475,3.461,-56.947,174.722,18.279,152.924
C06213=1087.480,3.711,-56.961,174.724,18.282,152.925
C06214=1087.486,3.961,-56.975,174.725,18.283,152.925
C06215=1087.492,4.210,-56.989,174.727,18.285,152.925
C06216=1087.497,4.460,-57.003,174.729,18.287,152.925
C06217=1087.504,4.709,-57.017,174.730,18.289,152.925
C06218=1087.509,4.958,-57.031,174.732,18.290,152.925
C06219=1087.515,5.209,-57.045,174.733,18.292,152.925
C06220=1087.521,5.458,-57.059,174.735,18.294,152.925
C06221=1087.526,5.708,-57.073,174.737,18.296,152.925
C06222=1087.532,5.957,-57.087,174.738,18.298,152.925
C06223=1087.539,6.207,-57.101,174.740,18.300,152.925
C06224=1087.544,6.456,-57.115,174.742,18.301,152.925
C06225=1087.550,6.706,-57.129,174.743,18.303,152.925
C06226=1087.555,6.955,-57.143,174.744,18.304,152.925
C06227=1087.561,7.205,-57.157,174.747,18.306,152.925
C06228=1087.567,7.455,-57.171,174.748,18.308,152.925
C06229=1087.573,7.704,-57.186,174.749,18.310,152.925
C06230=1087.578,7.953,-57.200,174.752,18.312,152.925
C06231=1087.585,8.203,-57.213,174.753,18.314,152.925
C06232=1087.591,8.452,-57.228,174.754,18.315,152.926
C06233=1087.596,8.702,-57.242,174.756,18.317,152.926
C06234=1087.602,8.951,-57.256,174.758,18.319,152.926
C06235=1087.608,9.201,-57.271,174.759,18.320,152.926
C06236=1087.614,9.450,-57.285,174.761,18.322,152.926
C06237=1087.619,9.700,-57.298,174.763,18.325,152.926
C06238=1087.625,9.950,-57.313,174.764,18.326,152.926
C06239=1087.631,10.199,-57.327,174.766,18.328,152.926
C06240=1087.637,10.448,-57.340,174.768,18.330,152.926
C06241=1087.644,10.698,-57.355,174.769,18.331,152.926
C06242=1087.649,10.948,-57.369,174.771,18.333,152.926
C06243=1087.655,11.197,-57.384,174.772,18.334,152.926
C06244=1087.661,11.447,-57.398,174.774,18.336,152.926
C06245=1087.666,11.697,-57.412,174.776,18.338,152.926
C06246=1087.672,11.945,-57.427,174.777,18.340,152.926
C06247=1087.678,12.196,-57.441,174.779,18.342,152.926
C06248=1087.684,12.445,-57.455,174.781,18.344,152.926
C06249=1087.689,12.694,-57.469,174.782,18.345,152.926
C06250=1087.696,12.944,-57.484,174.784,18.347,152.926
C06251=1087.701,13.194,-57.498,174.786,18.349,152.926
C06252=1087.707,13.442,-57.513,174.787,18.351,152.926
C06253=1087.713,13.693,-57.527,174.788,18.352,152.927
C06254=1087.719,13.942,-57.541,174.791,18.354,152.927
C06255=1087.725,14.192,-57.556,174.792,18.356,152.927
C06256=1087.731,14.441,-57.570,174.794,18.357,152.927
C06257=1087.736,14.691,-57.584,174.796,18.359,152.927
C06258=1087.743,14.967,-57.600,174.797,18.361,152.927
C06259=1087.750,15.243,-57.617,174.799,18.363,152.927
C06260=1087.757,15.518,-57.632,174.801,18.365,152.927
C06261=1087.763,15.795,-57.648,174.803,18.367,152.927
C06262=1087.767,16.044,-57.662,174.804,18.369,152.927
C06263=1087.773,16.293,-57.677,174.806,18.371,152.927
C06264=1087.780,16.543,-57.692,174.808,18.373,152.927
C06265=1087.785,16.793,-57.706,174.809,18.374,152.927
C06266=1087.792,17.042,-57.721,174.811,18.376,152.927
C06267=1087.797,17.292,-57.735,174.813,18.378,152.927
C06268=1087.803,17.541,-57.749,174.814,18.380,152.927
C06269=1087.808,17.791,-57.765,174.816,18.381,152.927
C06270=1087.814,18.040,-57.779,174.818,18.383,152.927
C06271=1087.820,18.289,-57.793,174.819,18.385,152.927
C06272=1087.826,18.540,-57.807,174.821,18.386,152.927
C06273=1087.832,18.789,-57.822,174.823,18.389,152.928
C06274=1087.838,19.038,-57.837,174.824,18.390,152.928
C06275=1087.843,19.288,-57.851,174.825,18.392,152.928
C06276=1087.848,19.537,-57.866,174.828,18.394,152.928
C06277=1087.855,19.787,-57.881,174.829,18.396,152.928
C06278=1087.860,20.036,-57.895,174.830,18.397,152.928
C06279=1087.867,20.286,-57.910,174.833,18.399,152.928
C06280=1087.872,20.535,-57.924,174.834,18.401,152.928
C06281=1087.878,20.785,-57.939,174.836,18.402,152.928
C06282=1087.884,21.034,-57.954,174.838,18.404,152.928
C06283=1087.889,21.283,-57.968,174.839,18.407,152.928
C06284=1087.895,21.533,-57.984,174.840,18.408,152.928
C06285=1087.900,21.783,-57.998,174.843,18.410,152.928
C06286=1087.907,22.033,-58.013,174.844,18.412,152.928
C06287=1087.913,22.282,-58.027,174.845,18.413,152.928
C06288=1087.918,22.531,-58.042,174.848,18.415,152.928
C06289=1087.924,22.781,-58.057,174.849,18.417,152.928
C06290=1087.930,23.030,-58.071,174.850,18.418,152.928
C06291=1087.935,23.280,-58.087,174.853,18.421,152.928
C06292=1087.941,23.529,-58.101,174.854,18.422,152.928
C06293=1087.947,23.779,-58.115,174.856,18.424,152.928
C06294=1087.952,24.028,-58.131,174.858,18.426,152.928
C06295=1087.958,24.278,-58.146,174.859,18.428,152.929
C06296=1087.964,24.527,-58.160,174.861,18.430,152.929
C06297=1087.971,24.777,-58.175,174.863,18.431,152.929
C06298=1087.976,25.026,-58.190,174.864,18.433,152.929
C06299=1087.982,25.276,-58.205,174.866,18.435,152.929
C06300=1087.988,25.525,-58.219,174.868,18.437,152.929
C06301=1087.993,25.775,-58.235,174.869,18.438,152.929
C06302=1087.999,26.024,-58.249,174.871,18.440,152.929
C06303=1088.005,26.274,-58.264,174.873,18.442,152.929
C06304=1088.010,26.523,-58.279,174.874,18.443,152.929
C06305=1088.017,26.773,-58.294,174.876,18.445,152.929
C06306=1088.022,27.023,-58.309,174.878,18.447,152.929
C06307=1088.028,27.272,-58.324,174.879,18.449,152.929
C06308=1088.034,27.521,-58.338,174.882,18.451,152.929
C06309=1088.039,27.771,-58.354,174.883,18.452,152.929
C06310=1088.045,28.020,-58.368,174.884,18.454,152.929
C06311=1088.051,28.270,-58.383,174.886,18.456,152.929
C06312=1088.057,28.519,-58.399,174.888,18.458,152.929
C06313=1088.063,28.769,-58.413,174.889,18.459,152.929
C06314=1088.068,29.018,-58.429,174.891,18.461,152.929
C06315=1088.074,29.268,-58.444,174.893,18.463,152.929
C06316=1088.079,29.517,-58.459,174.895,18.465,152.929
C06317=1088.086,29.767,-58.474,174.896,18.467,152.929
C06318=1088.091,30.016,-58.489,174.898,18.468,152.929
C06319=1088.097,30.266,-58.504,174.900,18.470,152.929
C06320=1088.102,30.515,-58.519,174.902,18.472,152.929
C06321=1088.109,30.764,-58.534,174.903,18.473,152.930
C06322=1088.115,31.042,-58.551,174.905,18.475,152.930
C06323=1088.121,31.319,-58.568,174.907,18.478,152.930
C06324=1088.127,31.596,-58.585,174.909,18.480,152.930
C06325=1088.133,31.874,-58.601,174.911,18.482,152.930
C06326=1088.140,32.123,-58.616,174.912,18.483,152.930
C06327=1088.145,32.373,-58.632,174.915,18.485,152.930
C06328=1088.151,32.622,-58.647,174.916,18.487,152.930
C06329=1088.157,32.872,-58.662,174.917,18.488,152.930
C06330=1088.162,33.121,-58.677,174.920,18.491,152.930
C06331=1088.168,33.371,-58.692,174.921,18.492,152.930
C06332=1088.173,33.620,-58.707,174.923,18.494,152.930
C06333=1088.180,33.870,-58.722,174.925,18.496,152.930
C06334=1088.185,34.120,-58.738,174.926,18.497,152.930
C06335=1088.191,34.369,-58.752,174.928,18.499,152.930
C06336=1088.197,34.618,-58.769,174.930,18.501,152.930
C06337=1088.202,34.867,-58.784,174.931,18.502,152.930
C06338=1088.209,35.117,-58.799,174.933,18.504,152.930
C06339=1088.214,35.367,-58.814,174.935,18.506,152.930
C06340=1088.220,35.616,-58.829,174.937,18.508,152.930
C06341=1088.226,35.866,-58.844,174.939,18.510,152.930
C06342=1088.232,36.114,-58.860,174.940,18.511,152.930
C06343=1088.237,36.364,-58.875,174.942,18.513,152.930
C06344=1088.243,36.614,-58.891,174.944,18.515,152.930
C06345=1088.249,36.863,-58.905,174.945,18.516,152.930
C06346=1088.254,37.113,-58.921,174.947,18.518,152.930
C06347=1088.261,37.362,-58.937,174.949,18.520,152.930
C06348=1088.266,37.612,-58.952,174.951,18.522,152.930
C06349=1088.272,37.861,-58.967,174.952,18.524,152.930
C06350=1088.278,38.111,-58.982,174.954,18.525,152.931
C06351=1088.284,38.360,-58.998,174.956,18.527,152.931
C06352=1088.289,38.610,-59.014,174.957,18.529,152.931
C06353=1088.294,38.859,-59.029,174.960,18.531,152.931
C06354=1088.301,39.109,-59.044,174.961,18.532,152.931
C06355=1088.307,39.358,-59.060,174.963,18.534,152.931
C06356=1088.312,39.607,-59.075,174.965,18.536,152.931
C06357=1088.317,39.857,-59.091,174.966,18.538,152.931
C06358=1088.324,40.106,-59.106,174.968,18.540,152.931
C06359=1088.329,40.356,-59.122,174.970,18.541,152.931
C06360=1088.335,40.606,-59.137,174.971,18.543,152.931
C06361=1088.341,40.855,-59.153,174.974,18.545,152.931
C06362=1088.346,41.104,-59.169,174.975,18.546,152.931
C06363=1088.352,41.354,-59.184,174.977,18.548,152.931
C06364=1088.358,41.603,-59.200,174.979,18.550,152.931
C06365=1088.363,41.852,-59.215,174.980,18.552,152.931
C06366=1088.369,42.102,-59.231,174.982,18.554,152.931
C06367=1088.375,42.352,-59.247,174.984,18.555,152.931
C06368=1088.380,42.601,-59.261,174.986,18.557,152.931
C06369=1088.386,42.851,-59.277,174.987,18.559,152.931
C06370=1088.392,43.100,-59.293,174.989,18.560,152.931
C06371=1088.397,43.349,-59.308,174.991,18.562,152.931
C06372=1088.403,43.599,-59.325,174.993,18.564,152.931
C06373=1088.409,43.848,-59.340,174.995,18.566,152.931
C06374=1088.415,44.098,-59.356,174.996,18.567,152.931
C06375=1088.420,44.347,-59.371,174.998,18.569,152.931
C06376=1088.426,44.597,-59.387,175.000,18.571,152.931
C06377=1088.431,44.846,-59.402,175.001,18.572,152.931
C06378=1088.437,45.095,-59.418,175.004,18.574,152.931
C06379=1088.443,45.345,-59.434,175.005,18.576,152.931
C06380=1088.449,45.595,-59.450,175.007,18.578,152.931
C06381=1088.454,45.843,-59.466,175.009,18.580,152.931
C06382=1088.460,46.093,-59.481,175.010,18.581,152.931
C06383=1088.466,46.343,-59.497,175.013,18.583,152.931
C06384=1088.471,46.592,-59.513,175.014,18.585,152.931
C06385=1088.477,46.841,-59.529,175.016,18.587,152.931
C06386=1088.482,47.119,-59.547,175.018,18.588,152.932
C06387=1088.489,47.396,-59.564,175.020,18.590,152.932
C06388=1088.495,47.674,-59.582,175.022,18.593,152.932
C06389=1088.502,47.951,-59.600,175.023,18.595,152.932
C06390=1088.507,48.201,-59.615,175.026,18.597,152.932
C06391=1088.513,48.450,-59.631,175.027,18.598,152.932
C06392=1088.518,48.700,-59.647,175.029,18.600,152.932
C06393=1088.524,48.949,-59.663,175.031,18.601,152.932
C06394=1088.530,49.198,-59.679,175.033,18.603,152.932
C06395=1088.535,49.448,-59.694,175.035,18.605,152.932
C06396=1088.541,49.697,-59.711,175.036,18.606,152.932
C06397=1088.547,49.947,-59.726,175.038,18.609,152.932
C06398=1088.552,50.196,-59.742,175.040,18.610,152.932
C06399=1088.558,50.445,-59.758,175.042,18.612,152.932
C06400=1088.564,50.695,-59.774,175.043,18.614,152.932
C06401=1088.570,50.944,-59.790,175.046,18.616,152.932
C06402=1088.575,51.194,-59.807,175.047,18.617,152.932
C06403=1088.580,51.443,-59.822,175.049,18.619,152.932
C06404=1088.586,51.693,-59.838,175.051,18.620,152.932
C06405=1088.592,51.942,-59.855,175.052,18.622,152.932
C06406=1088.598,52.192,-59.870,175.055,18.624,152.932
C06407=1088.603,52.441,-59.886,175.056,18.626,152.932
C06408=1088.609,52.690,-59.902,175.058,18.628,152.932
C06409=1088.615,52.939,-59.919,175.060,18.629,152.932
C06410=1088.620,53.189,-59.934,175.062,18.631,152.932
C06411=1088.626,53.439,-59.950,175.064,18.632,152.932
C06412=1088.632,53.688,-59.967,175.065,18.634,152.932
C06413=1088.638,53.937,-59.983,175.067,18.636,152.932
C06414=1088.643,54.187,-59.999,175.069,18.637,152.932
C06415=1088.649,54.436,-60.015,175.071,18.640,152.932
C06416=1088.654,54.686,-60.031,175.072,18.641,152.932
C06417=1088.660,54.935,-60.047,175.075,18.643,152.932
C06418=1088.666,55.184,-60.064,175.076,18.644,152.932
C06419=1088.672,55.434,-60.079,175.079,18.646,152.932
C06420=1088.678,55.684,-60.096,175.080,18.648,152.932
C06421=1088.683,55.932,-60.111,175.082,18.650,152.932
C06422=1088.689,56.182,-60.128,175.084,18.651,152.932
C06423=1088.695,56.431,-60.145,175.085,18.652,152.932
C06424=1088.700,56.681,-60.161,175.088,18.655,152.932
C06425=1088.706,56.931,-60.176,175.089,18.656,152.932
C06426=1088.712,57.180,-60.193,175.091,18.658,152.932
C06427=1088.718,57.429,-60.209,175.093,18.659,152.932
C06428=1088.724,57.679,-60.225,175.095,18.661,152.932
C06429=1088.729,57.928,-60.242,175.097,18.663,152.932
C06430=1088.735,58.178,-60.258,175.099,18.665,152.932
C06431=1088.741,58.427,-60.274,175.101,18.666,152.932
C06432=1088.747,58.676,-60.291,175.102,18.667,152.932
C06433=1088.752,58.925,-60.307,175.104,18.670,152.932
C06434=1088.758,59.174,-60.323,175.106,18.671,152.932
C06435=1088.764,59.424,-60.340,175.108,18.673,152.932
C06436=1088.769,59.673,-60.356,175.110,18.674,152.932
C06437=1088.775,59.923,-60.371,175.112,18.676,152.932
C06438=1088.781,60.173,-60.388,175.114,18.677,152.932
C06439=1088.787,60.422,-60.404,175.116,18.679,152.932
C06440=1088.792,60.672,-60.421,175.117,18.681,152.932
C06441=1088.798,60.921,-60.437,175.119,18.683,152.932
C06442=1088.804,61.170,-60.453,175.121,18.684,152.932
C06443=1088.810,61.420,-60.470,175.123,18.686,152.932
C06444=1088.816,61.669,-60.486,175.125,18.688,152.932
C06445=1088.822,61.918,-60.503,175.126,18.689,152.932
C06446=1088.828,62.167,-60.520,175.129,18.691,152.932
C06447=1088.833,62.417,-60.536,175.130,18.692,152.932
C06448=1088.839,62.666,-60.552,175.133,18.694,152.932
C06449=1088.845,62.916,-60.569,175.134,18.695,152.932
C06450=1088.852,63.193,-60.587,175.136,18.697,152.932
C06451=1088.858,63.471,-60.605,175.139,18.699,152.932
C06452=1088.865,63.748,-60.623,175.141,18.701,152.932
C06453=1088.871,64.025,-60.642,175.143,18.703,152.932
C06454=1088.877,64.275,-60.658,175.145,18.704,152.932
C06455=1088.882,64.524,-60.676,175.146,18.706,152.932
C06456=1088.888,64.773,-60.692,175.149,18.708,152.932
C06457=1088.894,65.022,-60.708,175.150,18.709,152.932
C06458=1088.900,65.272,-60.725,175.153,18.711,152.932
C06459=1088.906,65.521,-60.741,175.154,18.712,152.932
C06460=1088.911,65.771,-60.758,175.156,18.715,152.932
C06461=1088.917,66.020,-60.774,175.158,18.716,152.932
C06462=1088.922,66.269,-60.792,175.160,18.718,152.932
C06463=1088.928,66.519,-60.808,175.162,18.719,152.932
C06464=1088.934,66.768,-60.824,175.164,18.721,152.931
C06465=1088.939,67.018,-60.841,175.166,18.722,152.932
C06466=1088.945,67.267,-60.857,175.168,18.724,152.932
C06467=1088.951,67.516,-60.875,175.170,18.725,152.931
C06468=1088.957,67.765,-60.891,175.172,18.727,152.931
C06469=1088.962,68.015,-60.908,175.173,18.729,152.932
C06470=1088.968,68.264,-60.924,175.176,18.731,152.931
C06471=1088.973,68.513,-60.942,175.177,18.732,152.931
C06472=1088.979,68.763,-60.958,175.179,18.734,152.931
C06473=1088.985,69.012,-60.975,175.181,18.735,152.931
C06474=1088.991,69.262,-60.991,175.183,18.737,152.931
C06475=1088.996,69.511,-61.009,175.185,18.738,152.931
C06476=1089.002,69.760,-61.025,175.187,18.740,152.931
C06477=1089.007,70.010,-61.042,175.189,18.742,152.931
C06478=1089.014,70.259,-61.059,175.191,18.744,152.931
C06479=1089.019,70.509,-61.076,175.193,18.745,152.931
C06480=1089.025,70.758,-61.092,175.195,18.747,152.931
C06481=1089.031,71.007,-61.110,175.197,18.748,152.931
C06482=1089.036,71.257,-61.127,175.199,18.750,152.931
C06483=1089.042,71.506,-61.143,175.200,18.752,152.931
C06484=1089.047,71.755,-61.161,175.203,18.753,152.931
C06485=1089.053,72.005,-61.177,175.204,18.755,152.931
C06486=1089.059,72.254,-61.194,175.207,18.756,152.931
C06487=1089.064,72.503,-61.211,175.208,18.758,152.931
C06488=1089.070,72.753,-61.228,175.210,18.760,152.931
C06489=1089.076,73.002,-61.245,175.212,18.761,152.931
C06490=1089.081,73.251,-61.262,175.214,18.763,152.931
C06491=1089.087,73.502,-61.279,175.216,18.764,152.931
C06492=1089.093,73.751,-61.296,175.218,18.766,152.931
C06493=1089.099,74.000,-61.312,175.220,18.768,152.931
C06494=1089.104,74.249,-61.330,175.222,18.769,152.931
C06495=1089.110,74.499,-61.347,175.224,18.771,152.931
C06496=1089.116,74.747,-61.364,175.226,18.772,152.931
C06497=1089.121,74.997,-61.381,175.228,18.774,152.931
C06498=1089.127,75.246,-61.398,175.230,18.776,152.931
C06499=1089.133,75.496,-61.415,175.232,18.777,152.931
C06500=1089.139,75.745,-61.432,175.234,18.779,152.931
C06501=1089.144,75.995,-61.449,175.235,18.780,152.931
C06502=1089.149,76.244,-61.467,175.238,18.782,152.931
C06503=1089.155,76.493,-61.483,175.239,18.783,152.931
C06504=1089.161,76.742,-61.501,175.242,18.785,152.931
C06505=1089.166,76.992,-61.518,175.243,18.786,152.930
C06506=1089.173,77.241,-61.535,175.246,18.789,152.930
C06507=1089.178,77.491,-61.552,175.247,18.790,152.930
C06508=1089.184,77.740,-61.569,175.250,18.792,152.930
C06509=1089.190,77.989,-61.586,175.251,18.793,152.930
C06510=1089.195,78.238,-61.603,175.253,18.795,152.930
C06511=1089.201,78.488,-61.621,175.255,18.796,152.930
C06512=1089.206,78.738,-61.638,175.257,18.798,152.930
C06513=1089.212,78.987,-61.655,175.260,18.799,152.930
C06514=1089.218,79.264,-61.675,175.261,18.801,152.930
C06515=1089.225,79.541,-61.693,175.264,18.803,152.930
C06516=1089.230,79.818,-61.713,175.266,18.805,152.930
C06517=1089.237,80.095,-61.732,175.268,18.807,152.930
C06518=1089.243,80.344,-61.750,175.270,18.808,152.930
C06519=1089.248,80.594,-61.767,175.272,18.810,152.930
C06520=1089.254,80.844,-61.784,175.274,18.811,152.930
C06521=1089.260,81.092,-61.801,175.276,18.813,152.930
C06522=1089.265,81.342,-61.818,175.278,18.814,152.930
C06523=1089.271,81.591,-61.836,175.280,18.816,152.930
C06524=1089.276,81.840,-61.853,175.283,18.818,152.930
C06525=1089.282,82.091,-61.871,175.284,18.819,152.930
C06526=1089.288,82.340,-61.888,175.287,18.821,152.930
C06527=1089.293,82.589,-61.906,175.288,18.822,152.930
C06528=1089.299,82.838,-61.923,175.291,18.824,152.929
C06529=1089.304,83.087,-61.940,175.292,18.825,152.930
C06530=1089.310,83.337,-61.958,175.295,18.827,152.929
C06531=1089.316,83.586,-61.976,175.296,18.828,152.929
C06532=1089.322,83.835,-61.993,175.298,18.830,152.929
C06533=1089.327,84.084,-62.009,175.300,18.831,152.929
C06534=1089.333,84.334,-62.027,175.302,18.833,152.929
C06535=1089.339,84.583,-62.045,175.305,18.835,152.929
C06536=1089.344,84.832,-62.063,175.306,18.836,152.929
C06537=1089.350,85.081,-62.080,175.309,18.838,152.929
C06538=1089.356,85.332,-62.097,175.311,18.839,152.929
C06539=1089.361,85.581,-62.115,175.313,18.841,152.929
C06540=1089.367,85.830,-62.132,175.314,18.842,152.929
C06541=1089.373,86.080,-62.150,175.317,18.844,152.929
C06542=1089.378,86.329,-62.168,175.318,18.845,152.929
C06543=1089.384,86.578,-62.186,175.321,18.846,152.929
C06544=1089.389,86.827,-62.203,175.322,18.848,152.929
C06545=1089.395,87.076,-62.221,175.325,18.850,152.929
C06546=1089.401,87.326,-62.238,175.327,18.851,152.928
C06547=1089.406,87.575,-62.255,175.329,18.853,152.928
C06548=1089.412,87.825,-62.273,175.331,18.854,152.928
C06549=1089.418,88.074,-62.291,175.333,18.855,152.928
C06550=1089.423,88.323,-62.309,175.335,18.857,152.928
C06551=1089.429,88.573,-62.326,175.337,18.858,152.928
C06552=1089.435,88.822,-62.344,175.339,18.860,152.928
C06553=1089.440,89.071,-62.362,175.342,18.862,152.928
C06554=1089.447,89.320,-62.380,175.343,18.863,152.928
C06555=1089.452,89.570,-62.397,175.346,18.865,152.928
C06556=1089.458,89.819,-62.415,175.347,18.866,152.928
C06557=1089.464,90.068,-62.433,175.350,18.868,152.928
C06558=1089.469,90.317,-62.450,175.352,18.869,152.928
C06559=1089.475,90.567,-62.468,175.354,18.870,152.928
C06560=1089.481,90.816,-62.486,175.355,18.872,152.928
C06561=1089.486,91.065,-62.503,175.358,18.873,152.927
C06562=1089.492,91.315,-62.521,175.361,18.875,152.927
C06563=1089.497,91.564,-62.539,175.362,18.877,152.927
C06564=1089.503,91.813,-62.557,175.364,18.878,152.927
C06565=1089.509,92.063,-62.575,175.366,18.879,152.927
C06566=1089.514,92.312,-62.592,175.368,18.881,152.927
C06567=1089.520,92.561,-62.610,175.371,18.883,152.927
C06568=1089.526,92.811,-62.629,175.373,18.884,152.927
C06569=1089.531,93.060,-62.647,175.375,18.886,152.927
C06570=1089.537,93.309,-62.664,175.377,18.887,152.927
C06571=1089.543,93.558,-62.682,175.379,18.888,152.927
C06572=1089.548,93.808,-62.700,175.380,18.890,152.927
C06573=1089.554,94.057,-62.718,175.383,18.892,152.927
C06574=1089.559,94.306,-62.736,175.386,18.893,152.927
C06575=1089.565,94.555,-62.754,175.387,18.894,152.926
C06576=1089.570,94.805,-62.773,175.389,18.896,152.926
C06577=1089.576,95.054,-62.790,175.391,18.897,152.926
C06578=1089.582,95.332,-62.810,175.394,18.899,152.926
C06579=1089.589,95.609,-62.830,175.396,18.900,152.926
C06580=1089.595,95.885,-62.850,175.398,18.902,152.926
C06581=1089.601,96.163,-62.870,175.401,18.904,152.926
C06582=1089.607,96.412,-62.888,175.403,18.905,152.926
C06583=1089.613,96.662,-62.907,175.405,18.907,152.926
C06584=1089.618,96.911,-62.925,175.407,18.909,152.926
C06585=1089.624,97.160,-62.943,175.409,18.910,152.926
C06586=1089.630,97.409,-62.960,175.412,18.911,152.926
C06587=1089.635,97.658,-62.979,175.413,18.912,152.925
C06588=1089.641,97.908,-62.997,175.416,18.914,152.925
C06589=1089.646,98.157,-63.014,175.418,18.915,152.925
C06590=1089.652,98.406,-63.034,175.420,18.917,152.925
C06591=1089.658,98.655,-63.051,175.422,18.919,152.925
C06592=1089.664,98.905,-63.069,175.424,18.920,152.925
C06593=1089.669,99.154,-63.087,175.426,18.921,152.925
C06594=1089.675,99.404,-63.106,175.429,18.923,152.925
C06595=1089.680,99.653,-63.124,175.431,18.924,152.925
C06596=1089.687,99.902,-63.142,175.433,18.926,152.925
C06597=1089.692,100.151,-63.160,175.435,18.927,152.925
C06598=1089.698,100.401,-63.178,175.437,18.928,152.924
C06599=1089.704,100.649,-63.197,175.440,18.930,152.924
C06600=1089.709,100.899,-63.215,175.441,18.931,152.924
C06601=1089.715,101.148,-63.233,175.444,18.933,152.924
C06602=1089.720,101.398,-63.252,175.445,18.934,152.924
C06603=1089.726,101.647,-63.270,175.448,18.935,152.924
C06604=1089.732,101.896,-63.288,175.450,18.937,152.924
C06605=1089.737,102.145,-63.306,175.452,18.938,152.924
C06606=1089.743,102.395,-63.325,175.454,18.940,152.924
C06607=1089.748,102.644,-63.343,175.457,18.941,152.924
C06608=1089.754,102.894,-63.361,175.459,18.942,152.923
C06609=1089.759,103.142,-63.380,175.461,18.944,152.923
C06610=1089.765,103.392,-63.398,175.463,18.945,152.923
C06611=1089.771,103.641,-63.417,175.465,18.947,152.923
C06612=1089.776,103.891,-63.435,175.468,18.949,152.923
C06613=1089.782,104.139,-63.454,175.469,18.950,152.923
C06614=1089.787,104.389,-63.472,175.472,18.951,152.923
C06615=1089.793,104.638,-63.490,175.474,18.953,152.923
C06616=1089.798,104.888,-63.509,175.476,18.954,152.923
C06617=1089.804,105.136,-63.527,175.479,18.955,152.923
C06618=1089.810,105.386,-63.546,175.480,18.956,152.923
C06619=1089.816,105.635,-63.564,175.483,18.958,152.922
C06620=1089.821,105.884,-63.583,175.485,18.960,152.922
C06621=1089.827,106.134,-63.601,175.487,18.961,152.922
C06622=1089.832,106.383,-63.620,175.489,18.962,152.922
C06623=1089.838,106.633,-63.639,175.492,18.964,152.922
C06624=1089.843,106.881,-63.657,175.493,18.965,152.922
C06625=1089.849,107.131,-63.676,175.496,18.967,152.922
C06626=1089.855,107.380,-63.694,175.498,18.968,152.922
C06627=1089.860,107.629,-63.713,175.500,18.969,152.922
C06628=1089.867,107.878,-63.732,175.503,18.971,152.921
C06629=1089.872,108.127,-63.750,175.504,18.972,152.921
C06630=1089.877,108.377,-63.769,175.507,18.974,152.921
C06631=1089.884,108.626,-63.788,175.509,18.975,152.921
C06632=1089.888,108.875,-63.806,175.511,18.976,152.921
C06633=1089.895,109.124,-63.824,175.514,18.978,152.921
C06634=1089.900,109.373,-63.843,175.516,18.979,152.921
C06635=1089.905,109.623,-63.862,175.518,18.980,152.921
C06636=1089.912,109.872,-63.881,175.520,18.981,152.920
C06637=1089.917,110.121,-63.899,175.522,18.982,152.920
C06638=1089.923,110.371,-63.917,175.525,18.984,152.920
C06639=1089.929,110.620,-63.937,175.527,18.986,152.920
C06640=1089.934,110.869,-63.955,175.529,18.987,152.920
C06641=1089.940,111.118,-63.974,175.531,18.988,152.920
C06642=1089.946,111.396,-63.996,175.534,18.990,152.920
C06643=1089.953,111.673,-64.016,175.536,18.991,152.920
C06644=1089.959,111.950,-64.036,175.539,18.993,152.919
C06645=1089.965,112.228,-64.058,175.541,18.994,152.919
C06646=1089.971,112.477,-64.076,175.543,18.996,152.919
C06647=1089.976,112.726,-64.095,175.546,18.997,152.919
C06648=1089.982,112.975,-64.114,175.548,18.999,152.919
C06649=1089.987,113.224,-64.134,175.550,18.999,152.919
C06650=1089.993,113.473,-64.152,175.553,19.001,152.919
C06651=1089.999,113.723,-64.170,175.555,19.002,152.919
C06652=1090.004,113.972,-64.190,175.557,19.003,152.918
C06653=1090.010,114.222,-64.209,175.559,19.005,152.918
C06654=1090.016,114.470,-64.227,175.562,19.006,152.918
C06655=1090.022,114.720,-64.246,175.564,19.007,152.918
C06656=1090.027,114.969,-64.266,175.566,19.009,152.918
C06657=1090.032,115.218,-64.285,175.569,19.011,152.918
C06658=1090.038,115.467,-64.304,175.570,19.012,152.918
C06659=1090.043,115.716,-64.323,175.573,19.013,152.918
C06660=1090.049,115.965,-64.342,175.575,19.015,152.917
C06661=1090.054,116.215,-64.360,175.577,19.016,152.917
C06662=1090.059,116.464,-64.379,175.579,19.017,152.917
C06663=1090.065,116.714,-64.399,175.582,19.018,152.917
C06664=1090.071,116.963,-64.418,175.584,19.019,152.917
C06665=1090.076,117.213,-64.437,175.586,19.021,152.917
C06666=1090.081,117.461,-64.456,175.589,19.023,152.917
C06667=1090.087,117.711,-64.475,175.591,19.024,152.917
C06668=1090.093,117.960,-64.494,175.593,19.025,152.916
C06669=1090.098,118.209,-64.513,175.596,19.027,152.916
C06670=1090.104,118.458,-64.533,175.598,19.028,152.916
C06671=1090.109,118.708,-64.552,175.600,19.029,152.916
C06672=1090.115,118.955,-64.571,175.603,19.030,152.916
C06673=1090.121,119.205,-64.590,175.605,19.032,152.916
C06674=1090.127,119.454,-64.609,175.607,19.033,152.916
C06675=1090.132,119.704,-64.629,175.609,19.035,152.916
C06676=1090.138,119.953,-64.647,175.612,19.036,152.915
C06677=1090.143,120.202,-64.667,175.614,19.037,152.915
C06678=1090.149,120.451,-64.686,175.616,19.038,152.915
C06679=1090.155,120.701,-64.705,175.619,19.040,152.915
C06680=1090.160,120.950,-64.724,175.620,19.041,152.915
C06681=1090.165,121.199,-64.743,175.623,19.042,152.915
C06682=1090.171,121.448,-64.764,175.625,19.044,152.915
C06683=1090.176,121.698,-64.783,175.627,19.045,152.914
C06684=1090.182,121.947,-64.802,175.630,19.046,152.914
C06685=1090.187,122.196,-64.821,175.632,19.048,152.914
C06686=1090.193,122.445,-64.840,175.635,19.049,152.914
C06687=1090.198,122.695,-64.860,175.637,19.050,152.914
C06688=1090.204,122.943,-64.880,175.639,19.051,152.914
C06689=1090.210,123.193,-64.899,175.642,19.053,152.913
C06690=1090.215,123.442,-64.918,175.644,19.054,152.913
C06691=1090.221,123.691,-64.937,175.646,19.055,152.913
C06692=1090.227,123.940,-64.957,175.649,19.057,152.913
C06693=1090.233,124.189,-64.976,175.651,19.058,152.913
C06694=1090.238,124.439,-64.995,175.653,19.059,152.913
C06695=1090.244,124.688,-65.015,175.656,19.060,152.912
C06696=1090.250,124.937,-65.035,175.658,19.062,152.912
C06697=1090.255,125.186,-65.053,175.660,19.062,152.912
C06698=1090.261,125.435,-65.073,175.663,19.064,152.912
C06699=1090.267,125.684,-65.093,175.665,19.065,152.912
C06700=1090.272,125.934,-65.113,175.667,19.066,152.912
C06701=1090.277,126.183,-65.132,175.670,19.068,152.912
C06702=1090.283,126.432,-65.152,175.672,19.069,152.911
C06703=1090.289,126.681,-65.171,175.675,19.070,152.911
C06704=1090.295,126.931,-65.190,175.677,19.071,152.911
C06705=1090.301,127.180,-65.210,175.679,19.073,152.911
C06706=1090.307,127.457,-65.232,175.682,19.074,152.911
C06707=1090.313,127.734,-65.254,175.685,19.075,152.911
C06708=1090.320,128.011,-65.275,175.687,19.077,152.910
C06709=1090.326,128.288,-65.297,175.690,19.078,152.910
C06710=1090.332,128.538,-65.316,175.693,19.079,152.910
C06711=1090.337,128.787,-65.337,175.694,19.080,152.910
C06712=1090.343,129.036,-65.356,175.697,19.082,152.910
C06713=1090.349,129.285,-65.376,175.700,19.083,152.909
C06714=1090.354,129.535,-65.395,175.702,19.084,152.909
C06715=1090.360,129.783,-65.415,175.704,19.085,152.909
C06716=1090.366,130.033,-65.434,175.707,19.087,152.909
C06717=1090.371,130.281,-65.454,175.709,19.088,152.909
C06718=1090.376,130.531,-65.474,175.712,19.089,152.909
C06719=1090.382,130.779,-65.494,175.714,19.090,152.908
C06720=1090.388,131.029,-65.513,175.716,19.091,152.908
C06721=1090.394,131.278,-65.533,175.719,19.092,152.908
C06722=1090.400,131.527,-65.552,175.721,19.093,152.908
C06723=1090.405,131.776,-65.573,175.723,19.094,152.908
C06724=1090.411,132.026,-65.592,175.726,19.096,152.907
C06725=1090.417,132.275,-65.612,175.729,19.097,152.907
C06726=1090.422,132.524,-65.631,175.730,19.098,152.907
C06727=1090.428,132.773,-65.652,175.733,19.099,152.907
C06728=1090.434,133.022,-65.672,175.736,19.101,152.907
C06729=1090.439,133.271,-65.691,175.738,19.102,152.907
C06730=1090.444,133.520,-65.711,175.740,19.103,152.906
C06731=1090.450,133.770,-65.731,175.743,19.104,152.906
C06732=1090.455,134.019,-65.751,175.745,19.105,152.906
C06733=1090.461,134.268,-65.771,175.748,19.107,152.906
C06734=1090.467,134.517,-65.790,175.750,19.108,152.906
C06735=1090.472,134.766,-65.811,175.752,19.109,152.905
C06736=1090.478,135.015,-65.831,175.755,19.110,152.905
C06737=1090.483,135.265,-65.851,175.758,19.112,152.905
C06738=1090.489,135.514,-65.871,175.760,19.112,152.905
C06739=1090.495,135.763,-65.891,175.762,19.114,152.905
C06740=1090.501,136.012,-65.911,175.765,19.115,152.904
C06741=1090.506,136.261,-65.930,175.767,19.117,152.904
C06742=1090.511,136.510,-65.951,175.769,19.117,152.904
C06743=1090.517,136.759,-65.971,175.772,19.119,152.904
C06744=1090.523,137.008,-65.990,175.775,19.120,152.904
C06745=1090.528,137.258,-66.011,175.777,19.121,152.904
C06746=1090.534,137.506,-66.031,175.779,19.122,152.903
C06747=1090.540,137.756,-66.051,175.782,19.123,152.903
C06748=1090.546,138.005,-66.072,175.784,19.124,152.903
C06749=1090.551,138.255,-66.091,175.787,19.126,152.903
C06750=1090.557,138.504,-66.111,175.789,19.127,152.903
C06751=1090.562,138.753,-66.132,175.792,19.128,152.902
C06752=1090.568,139.002,-66.152,175.794,19.129,152.902
C06753=1090.574,139.251,-66.172,175.797,19.130,152.902
C06754=1090.580,139.499,-66.192,175.800,19.131,152.902
C06755=1090.585,139.749,-66.212,175.801,19.132,152.902
C06756=1090.591,139.998,-66.232,175.804,19.133,152.901
C06757=1090.596,140.247,-66.253,175.807,19.135,152.901
C06758=1090.602,140.496,-66.273,175.809,19.136,152.901
C06759=1090.607,140.745,-66.293,175.811,19.137,152.901
C06760=1090.612,140.994,-66.314,175.814,19.138,152.901
C06761=1090.618,141.243,-66.334,175.817,19.139,152.900
C06762=1090.624,141.493,-66.355,175.819,19.141,152.900
C06763=1090.630,141.742,-66.375,175.822,19.142,152.900
C06764=1090.636,141.991,-66.395,175.824,19.142,152.900
C06765=1090.640,142.241,-66.415,175.826,19.144,152.900
C06766=1090.646,142.489,-66.435,175.829,19.145,152.899
C06767=1090.652,142.738,-66.456,175.832,19.146,152.899
C06768=1090.657,142.988,-66.476,175.833,19.147,152.899
C06769=1090.663,143.236,-66.496,175.836,19.148,152.899
C06770=1090.669,143.514,-66.520,175.839,19.150,152.899
C06771=1090.676,143.791,-66.542,175.841,19.151,152.898
C06772=1090.682,144.068,-66.564,175.845,19.153,152.898
C06773=1090.688,144.346,-66.587,175.848,19.154,152.898
C06774=1090.694,144.594,-66.609,175.850,19.155,152.898
C06775=1090.700,144.843,-66.629,175.852,19.156,152.897
C06776=1090.705,145.092,-66.649,175.855,19.157,152.897
C06777=1090.710,145.341,-66.670,175.858,19.158,152.897
C06778=1090.716,145.590,-66.690,175.860,19.159,152.897
C06779=1090.722,145.840,-66.711,175.862,19.160,152.897
C06780=1090.727,146.089,-66.731,175.865,19.161,152.896
C06781=1090.733,146.338,-66.751,175.868,19.163,152.896
C06782=1090.738,146.587,-66.772,175.870,19.164,152.896
C06783=1090.744,146.836,-66.792,175.873,19.165,152.896
C06784=1090.749,147.085,-66.813,175.875,19.165,152.895
C06785=1090.756,147.334,-66.834,175.878,19.167,152.895
C06786=1090.761,147.583,-66.854,175.880,19.168,152.895
C06787=1090.766,147.832,-66.875,175.883,19.169,152.895
C06788=1090.772,148.081,-66.895,175.886,19.170,152.894
C06789=1090.779,148.330,-66.917,175.888,19.172,152.894
C06790=1090.784,148.579,-66.937,175.890,19.172,152.894
C06791=1090.789,148.829,-66.958,175.893,19.173,152.894
C06792=1090.794,149.078,-66.978,175.896,19.174,152.894
C06793=1090.800,149.327,-66.999,175.898,19.176,152.893
C06794=1090.806,149.576,-67.020,175.901,19.177,152.893
C06795=1090.812,149.825,-67.040,175.903,19.178,152.893
C06796=1090.817,150.074,-67.061,175.906,19.179,152.893
C06797=1090.822,150.323,-67.081,175.909,19.180,152.892
C06798=1090.828,150.572,-67.103,175.911,19.181,152.892
C06799=1090.834,150.821,-67.124,175.914,19.182,152.892
C06800=1090.839,151.071,-67.144,175.917,19.183,152.892
C06801=1090.844,151.319,-67.165,175.918,19.184,152.892
C06802=1090.851,151.569,-67.186,175.921,19.186,152.891
C06803=1090.856,151.818,-67.206,175.924,19.187,152.891
C06804=1090.862,152.066,-67.228,175.927,19.188,152.891
C06805=1090.867,152.315,-67.248,175.929,19.189,152.891
C06806=1090.873,152.565,-67.269,175.932,19.190,152.890
C06807=1090.879,152.814,-67.290,175.934,19.191,152.890
C06808=1090.884,153.063,-67.311,175.937,19.192,152.890
C06809=1090.889,153.311,-67.332,175.939,19.193,152.890
C06810=1090.895,153.561,-67.353,175.942,19.194,152.890
C06811=1090.900,153.810,-67.374,175.945,19.195,152.889
C06812=1090.906,154.059,-67.395,175.948,19.196,152.889
C06813=1090.912,154.309,-67.416,175.949,19.197,152.889
C06814=1090.917,154.557,-67.437,175.952,19.198,152.889
C06815=1090.923,154.806,-67.458,175.955,19.199,152.888
C06816=1090.929,155.055,-67.479,175.958,19.201,152.888
C06817=1090.934,155.304,-67.500,175.960,19.202,152.888
C06818=1090.940,155.553,-67.521,175.963,19.203,152.888
C06819=1090.946,155.803,-67.542,175.965,19.203,152.887
C06820=1090.951,156.051,-67.563,175.968,19.204,152.887
C06821=1090.956,156.300,-67.584,175.971,19.205,152.887
C06822=1090.963,156.550,-67.605,175.973,19.207,152.887
C06823=1090.968,156.799,-67.626,175.976,19.208,152.886
C06824=1090.973,157.047,-67.647,175.979,19.209,152.886
C06825=1090.979,157.297,-67.668,175.981,19.210,152.886
C06826=1090.985,157.546,-67.690,175.983,19.211,152.886
C06827=1090.990,157.794,-67.711,175.986,19.212,152.885
C06828=1090.996,158.044,-67.732,175.989,19.213,152.885
C06829=1091.001,158.293,-67.754,175.992,19.214,152.885
C06830=1091.006,158.542,-67.774,175.994,19.215,152.885
C06831=1091.012,158.791,-67.796,175.997,19.216,152.884
C06832=1091.018,159.040,-67.817,176.000,19.217,152.884
C06833=1091.024,159.289,-67.838,176.003,19.218,152.884
C06834=1091.030,159.566,-67.861,176.005,19.219,152.884
C06835=1091.036,159.843,-67.885,176.008,19.220,152.883
C06836=1091.042,160.119,-67.909,176.011,19.222,152.883
C06837=1091.049,160.396,-67.932,176.014,19.223,152.883
C06838=1091.054,160.646,-67.954,176.016,19.224,152.883
C06839=1091.059,160.894,-67.975,176.019,19.225,152.882
C06840=1091.066,161.144,-67.997,176.022,19.226,152.882
C06841=1091.071,161.392,-68.018,176.025,19.227,152.882
C06842=1091.077,161.642,-68.039,176.027,19.228,152.882
C06843=1091.082,161.891,-68.061,176.030,19.229,152.881
C06844=1091.087,162.139,-68.082,176.032,19.230,152.881
C06845=1091.093,162.389,-68.103,176.035,19.231,152.881
C06846=1091.098,162.638,-68.125,176.038,19.232,152.881
C06847=1091.104,162.886,-68.146,176.040,19.233,152.880
C06848=1091.109,163.136,-68.168,176.043,19.234,152.880
C06849=1091.115,163.384,-68.190,176.046,19.236,152.880
C06850=1091.121,163.634,-68.211,176.048,19.237,152.880
C06851=1091.125,163.883,-68.232,176.051,19.238,152.879
C06852=1091.131,164.132,-68.254,176.054,19.239,152.879
C06853=1091.136,164.381,-68.276,176.057,19.240,152.879
C06854=1091.142,164.630,-68.297,176.059,19.240,152.879
C06855=1091.148,164.879,-68.319,176.061,19.242,152.878
C06856=1091.153,165.128,-68.341,176.064,19.243,152.878
C06857=1091.158,165.377,-68.361,176.067,19.244,152.878
C06858=1091.164,165.626,-68.383,176.070,19.245,152.878
C06859=1091.169,165.875,-68.405,176.072,19.246,152.877
C06860=1091.175,166.124,-68.427,176.075,19.247,152.877
C06861=1091.180,166.373,-68.448,176.078,19.248,152.877
C06862=1091.186,166.622,-68.470,176.081,19.249,152.877
C06863=1091.191,166.871,-68.492,176.084,19.250,152.876
C06864=1091.197,167.120,-68.513,176.086,19.251,152.876
C06865=1091.202,167.369,-68.535,176.088,19.252,152.876
C06866=1091.208,167.617,-68.556,176.091,19.253,152.876
C06867=1091.213,167.867,-68.579,176.094,19.254,152.875
C06868=1091.219,168.115,-68.600,176.097,19.255,152.875
C06869=1091.224,168.365,-68.622,176.099,19.256,152.875
C06870=1091.230,168.613,-68.643,176.102,19.257,152.875
C06871=1091.235,168.863,-68.666,176.105,19.258,152.874
C06872=1091.241,169.111,-68.687,176.108,19.259,152.874
C06873=1091.246,169.361,-68.709,176.110,19.260,152.874
C06874=1091.252,169.610,-68.731,176.113,19.262,152.873
C06875=1091.257,169.859,-68.753,176.116,19.263,152.873
C06876=1091.263,170.108,-68.774,176.119,19.264,152.873
C06877=1091.268,170.356,-68.797,176.121,19.265,152.873
C06878=1091.274,170.606,-68.819,176.124,19.265,152.872
C06879=1091.279,170.854,-68.840,176.126,19.266,152.872
C06880=1091.285,171.104,-68.862,176.129,19.267,152.872
C06881=1091.290,171.352,-68.884,176.132,19.268,152.872
C06882=1091.296,171.602,-68.906,176.135,19.269,152.871
C06883=1091.302,171.851,-68.928,176.137,19.270,152.871
C06884=1091.307,172.099,-68.950,176.140,19.271,152.871
C06885=1091.313,172.348,-68.972,176.143,19.272,152.871
C06886=1091.318,172.597,-68.994,176.146,19.273,152.870
C06887=1091.324,172.847,-69.016,176.149,19.274,152.870
C06888=1091.329,173.095,-69.037,176.151,19.275,152.870
C06889=1091.335,173.344,-69.060,176.154,19.276,152.869
C06890=1091.341,173.593,-69.082,176.157,19.277,152.869
C06891=1091.346,173.842,-69.104,176.160,19.278,152.869
C06892=1091.352,174.091,-69.125,176.163,19.279,152.868
C06893=1091.358,174.340,-69.148,176.165,19.280,152.868
C06894=1091.363,174.589,-69.170,176.168,19.281,152.868
C06895=1091.369,174.838,-69.192,176.170,19.282,152.868
C06896=1091.374,175.087,-69.215,176.173,19.282,152.867
C06897=1091.380,175.336,-69.236,176.176,19.283,152.867
C06898=1091.387,175.612,-69.261,176.180,19.285,152.867
C06899=1091.392,175.889,-69.285,176.183,19.286,152.866
C06900=1091.399,176.166,-69.310,176.185,19.287,152.866
C06901=1091.405,176.442,-69.334,176.189,19.288,152.866
C06902=1091.410,176.691,-69.356,176.191,19.288,152.865
C06903=1091.416,176.940,-69.379,176.194,19.290,152.865
C06904=1091.422,177.189,-69.401,176.197,19.291,152.865
C06905=1091.427,177.438,-69.423,176.200,19.291,152.865
C06906=1091.433,177.687,-69.446,176.202,19.292,152.864
C06907=1091.439,177.936,-69.467,176.205,19.293,152.864
C06908=1091.444,178.184,-69.490,176.208,19.295,152.864
C06909=1091.449,178.434,-69.512,176.211,19.295,152.863
C06910=1091.456,178.682,-69.535,176.214,19.296,152.863
C06911=1091.461,178.932,-69.557,176.216,19.297,152.863
C06912=1091.467,179.180,-69.579,176.219,19.298,152.862
C06913=1091.473,179.429,-69.601,176.222,19.299,152.862
C06914=1091.478,179.678,-69.624,176.225,19.300,152.862
C06915=1091.484,179.928,-69.646,176.228,19.301,152.862
C06916=1091.490,180.176,-69.668,176.231,19.302,152.861
C06917=1091.495,180.425,-69.690,176.234,19.302,152.861
C06918=1091.501,180.674,-69.713,176.236,19.303,152.861
C06919=1091.507,180.923,-69.735,176.239,19.305,152.860
C06920=1091.513,181.172,-69.758,176.242,19.305,152.860
C06921=1091.518,181.420,-69.781,176.245,19.306,152.860
C06922=1091.523,181.670,-69.803,176.248,19.307,152.859
C06923=1091.530,181.918,-69.825,176.251,19.308,152.859
C06924=1091.535,182.168,-69.847,176.253,19.309,152.859
C06925=1091.541,182.417,-69.870,176.257,19.310,152.858
C06926=1091.547,182.666,-69.893,176.259,19.311,152.858
C06927=1091.552,182.914,-69.915,176.262,19.311,152.858
C06928=1091.558,183.163,-69.937,176.265,19.312,152.857
C06929=1091.564,183.412,-69.960,176.268,19.313,152.857
C06930=1091.569,183.662,-69.983,176.271,19.314,152.857
C06931=1091.576,183.910,-70.005,176.274,19.315,152.857
C06932=1091.581,184.159,-70.028,176.277,19.316,152.856
C06933=1091.587,184.409,-70.050,176.279,19.317,152.856
C06934=1091.592,184.657,-70.073,176.282,19.317,152.856
C06935=1091.598,184.905,-70.095,176.285,19.319,152.855
C06936=1091.604,185.154,-70.118,176.288,19.319,152.855
C06937=1091.609,185.404,-70.140,176.291,19.320,152.855
C06938=1091.615,185.653,-70.163,176.294,19.321,152.854
C06939=1091.621,185.902,-70.186,176.297,19.322,152.854
C06940=1091.625,186.150,-70.209,176.299,19.323,152.854
C06941=1091.631,186.399,-70.232,176.302,19.324,152.853
C06942=1091.636,186.648,-70.255,176.305,19.325,152.853
C06943=1091.642,186.897,-70.277,176.308,19.326,152.853
C06944=1091.647,187.146,-70.300,176.311,19.327,152.853
C06945=1091.653,187.394,-70.323,176.313,19.328,152.852
C06946=1091.659,187.643,-70.346,176.316,19.329,152.852
C06947=1091.665,187.892,-70.369,176.319,19.330,152.852
C06948=1091.670,188.142,-70.391,176.322,19.331,152.851
C06949=1091.675,188.391,-70.415,176.325,19.331,152.851
C06950=1091.680,188.639,-70.437,176.328,19.333,152.851
C06951=1091.686,188.888,-70.460,176.330,19.334,152.850
C06952=1091.692,189.137,-70.483,176.334,19.335,152.850
C06953=1091.697,189.386,-70.506,176.337,19.336,152.850
C06954=1091.703,189.635,-70.529,176.340,19.337,152.850
C06955=1091.709,189.884,-70.552,176.343,19.338,152.849
C06956=1091.713,190.132,-70.575,176.346,19.339,152.849
C06957=1091.719,190.381,-70.598,176.348,19.340,152.849
C06958=1091.725,190.630,-70.621,176.351,19.340,152.848
C06959=1091.730,190.879,-70.644,176.354,19.341,152.848
C06960=1091.736,191.128,-70.667,176.357,19.342,152.848
C06961=1091.741,191.377,-70.690,176.360,19.343,152.847
C06962=1091.748,191.653,-70.716,176.363,19.344,152.847
C06963=1091.754,191.929,-70.741,176.366,19.345,152.847
C06964=1091.760,192.206,-70.766,176.369,19.346,152.846
C06965=1091.766,192.481,-70.792,176.373,19.348,152.846
C06966=1091.771,192.730,-70.815,176.376,19.348,152.846
C06967=1091.777,192.979,-70.838,176.379,19.349,152.845
C06968=1091.782,193.228,-70.862,176.382,19.350,152.845
C06969=1091.788,193.477,-70.885,176.385,19.351,152.845
C06970=1091.794,193.726,-70.908,176.388,19.352,152.844
C06971=1091.799,193.975,-70.931,176.390,19.353,152.844
C06972=1091.804,194.224,-70.954,176.393,19.353,152.844
C06973=1091.810,194.473,-70.977,176.396,19.354,152.843
C06974=1091.816,194.722,-71.000,176.399,19.355,152.843
C06975=1091.822,194.970,-71.024,176.402,19.356,152.843
C06976=1091.827,195.219,-71.048,176.405,19.357,152.842
C06977=1091.833,195.468,-71.070,176.408,19.358,152.842
C06978=1091.838,195.717,-71.093,176.410,19.359,152.842
C06979=1091.844,195.966,-71.116,176.414,19.360,152.841
C06980=1091.849,196.214,-71.141,176.417,19.361,152.841
C06981=1091.855,196.463,-71.164,176.420,19.362,152.841
C06982=1091.861,196.712,-71.186,176.423,19.362,152.840
C06983=1091.866,196.961,-71.211,176.426,19.363,152.840
C06984=1091.872,197.210,-71.234,176.429,19.364,152.840
C06985=1091.878,197.458,-71.257,176.432,19.365,152.839
C06986=1091.883,197.707,-71.280,176.435,19.366,152.839
C06987=1091.889,197.956,-71.304,176.437,19.367,152.839
C06988=1091.895,198.206,-71.327,176.440,19.368,152.838
C06989=1091.901,198.454,-71.350,176.443,19.369,152.838
C06990=1091.906,198.703,-71.374,176.447,19.370,152.838
C06991=1091.912,198.952,-71.397,176.450,19.370,152.837
C06992=1091.918,199.201,-71.420,176.453,19.371,152.837
C06993=1091.923,199.449,-71.445,176.456,19.372,152.837
C06994=1091.929,199.698,-71.467,176.458,19.373,152.836
C06995=1091.935,199.947,-71.491,176.461,19.374,152.836
C06996=1091.940,200.196,-71.515,176.464,19.374,152.836
C06997=1091.945,200.445,-71.538,176.467,19.376,152.835
C06998=1091.951,200.694,-71.562,176.470,19.376,152.835
C06999=1091.957,200.943,-71.585,176.473,19.377,152.835
C07000=1091.963,201.191,-71.609,176.477,19.378,152.834
C07001=1091.968,201.440,-71.632,176.480,19.379,152.834
C07002=1091.974,201.689,-71.656,176.483,19.380,152.834
C07003=1091.980,201.938,-71.679,176.486,19.381,152.833
C07004=1091.985,202.186,-71.703,176.489,19.381,152.833
C07005=1091.991,202.436,-71.727,176.491,19.382,152.833
C07006=1091.997,202.684,-71.751,176.494,19.383,152.832
C07007=1092.002,202.933,-71.774,176.497,19.384,152.832
C07008=1092.008,203.182,-71.798,176.501,19.385,152.832
C07009=1092.014,203.430,-71.822,176.504,19.386,152.831
C07010=1092.019,203.679,-71.845,176.507,19.387,152.831
C07011=1092.025,203.928,-71.869,176.510,19.388,152.831
C07012=1092.030,204.177,-71.893,176.512,19.389,152.830
C07013=1092.036,204.426,-71.917,176.515,19.389,152.830
C07014=1092.042,204.674,-71.941,176.518,19.390,152.830
C07015=1092.047,204.924,-71.964,176.522,19.392,152.829
C07016=1092.053,205.172,-71.988,176.525,19.393,152.829
C07017=1092.058,205.421,-72.011,176.528,19.393,152.829
C07018=1092.063,205.670,-72.036,176.531,19.394,152.828
C07019=1092.070,205.919,-72.060,176.534,19.395,152.828
C07020=1092.075,206.168,-72.083,176.537,19.396,152.828
C07021=1092.080,206.416,-72.108,176.539,19.397,152.827
C07022=1092.086,206.665,-72.131,176.543,19.398,152.827
C07023=1092.091,206.913,-72.155,176.546,19.399,152.827
C07024=1092.098,207.163,-72.179,176.549,19.400,152.826
C07025=1092.103,207.411,-72.203,176.552,19.400,152.826
C07026=1092.126,208.430,-72.301,176.613,19.429,152.821
C07027=1092.135,208.808,-72.338,176.618,19.433,152.821
C07028=1092.143,209.186,-72.375,176.623,19.435,152.821
C07029=1092.152,209.564,-72.412,176.627,19.438,152.821
C07030=1092.160,209.941,-72.449,176.631,19.440,152.821
C07031=1092.165,210.190,-72.473,176.634,19.443,152.821
C07032=1092.171,210.439,-72.498,176.637,19.444,152.820
C07033=1092.176,210.688,-72.522,176.640,19.446,152.820
C07034=1092.182,210.937,-72.547,176.643,19.447,152.820
C07035=1092.188,211.186,-72.571,176.646,19.449,152.820
C07036=1092.193,211.434,-72.596,176.649,19.451,152.820
C07037=1092.199,211.683,-72.621,176.651,19.453,152.820
C07038=1092.204,211.932,-72.645,176.655,19.455,152.820
C07039=1092.210,212.180,-72.669,176.657,19.456,152.820
C07040=1092.216,212.429,-72.693,176.661,19.458,152.819
C07041=1092.222,212.678,-72.717,176.663,19.460,152.819
C07042=1092.228,212.926,-72.743,176.666,19.462,152.819
C07043=1092.233,213.175,-72.767,176.669,19.464,152.819
C07044=1092.238,213.424,-72.791,176.672,19.466,152.819
C07045=1092.244,213.673,-72.816,176.675,19.467,152.819
C07046=1092.249,213.921,-72.841,176.678,19.469,152.819
C07047=1092.255,214.170,-72.866,176.681,19.471,152.819
C07048=1092.260,214.419,-72.890,176.684,19.473,152.818
C07049=1092.266,214.668,-72.915,176.687,19.475,152.818
C07050=1092.272,214.916,-72.940,176.689,19.476,152.818
C07051=1092.277,215.165,-72.964,176.692,19.478,152.818
C07052=1092.283,215.414,-72.989,176.695,19.480,152.818
C07053=1092.289,215.662,-73.014,176.698,19.482,152.818
C07054=1092.294,215.912,-73.039,176.701,19.484,152.818
C07055=1092.299,216.160,-73.063,176.704,19.486,152.818
C07056=1092.305,216.409,-73.089,176.707,19.487,152.818
C07057=1092.311,216.658,-73.113,176.710,19.489,152.817
C07058=1092.317,216.906,-73.138,176.713,19.491,152.817
C07059=1092.322,217.155,-73.162,176.716,19.493,152.817
C07060=1092.328,217.403,-73.188,176.718,19.495,152.817
C07061=1092.333,217.652,-73.213,176.722,19.497,152.817
C07062=1092.339,217.902,-73.237,176.724,19.498,152.817
C07063=1092.344,218.150,-73.262,176.728,19.501,152.817
C07064=1092.350,218.399,-73.287,176.730,19.502,152.817
C07065=1092.356,218.647,-73.312,176.734,19.504,152.817
C07066=1092.362,218.896,-73.336,176.736,19.506,152.817
C07067=1092.367,219.144,-73.362,176.739,19.508,152.816
C07068=1092.373,219.394,-73.387,176.742,19.510,152.816
C07069=1092.378,219.642,-73.412,176.745,19.512,152.816
C07070=1092.384,219.891,-73.436,176.748,19.513,152.816
C07071=1092.389,220.139,-73.462,176.751,19.515,152.816
C07072=1092.395,220.388,-73.487,176.754,19.517,152.816
C07073=1092.401,220.637,-73.512,176.757,19.519,152.816
C07074=1092.407,220.885,-73.537,176.760,19.521,152.816
C07075=1092.413,221.134,-73.561,176.763,19.523,152.815
C07076=1092.417,221.383,-73.587,176.765,19.524,152.815
C07077=1092.424,221.631,-73.612,176.769,19.526,152.815
C07078=1092.429,221.880,-73.636,176.771,19.528,152.815
C07079=1092.438,222.262,-73.675,176.776,19.531,152.815
C07080=1092.446,222.643,-73.714,176.781,19.534,152.815
C07081=1092.455,223.025,-73.753,176.785,19.536,152.815
C07082=1092.463,223.406,-73.792,176.790,19.540,152.814
C07083=1092.470,223.655,-73.817,176.792,19.541,152.814
C07084=1092.474,223.904,-73.842,176.796,19.543,152.814
C07085=1092.480,224.153,-73.867,176.798,19.545,152.814
C07086=1092.485,224.401,-73.893,176.802,19.547,152.814
C07087=1092.491,224.650,-73.918,176.804,19.548,152.814
C07088=1092.497,224.899,-73.944,176.807,19.551,152.814
C07089=1092.502,225.147,-73.969,176.811,19.553,152.814
C07090=1092.508,225.396,-73.994,176.813,19.554,152.814
C07091=1092.514,225.645,-74.020,176.817,19.556,152.813
C07092=1092.519,225.893,-74.045,176.819,19.558,152.813
C07093=1092.525,226.142,-74.071,176.823,19.560,152.813
C07094=1092.531,226.391,-74.095,176.825,19.562,152.813
C07095=1092.536,226.639,-74.121,176.828,19.564,152.813
C07096=1092.542,226.888,-74.146,176.831,19.565,152.813
C07097=1092.547,227.137,-74.172,176.834,19.567,152.813
C07098=1092.553,227.385,-74.197,176.837,19.569,152.813
C07099=1092.558,227.634,-74.223,176.840,19.571,152.813
C07100=1092.565,227.883,-74.248,176.844,19.573,152.812
C07101=1092.570,228.132,-74.274,176.846,19.575,152.812
C07102=1092.576,228.380,-74.299,176.849,19.577,152.812
C07103=1092.581,228.629,-74.325,176.852,19.578,152.812
C07104=1092.587,228.877,-74.351,176.855,19.581,152.812
C07105=1092.592,229.125,-74.376,176.858,19.582,152.812
C07106=1092.598,229.374,-74.402,176.861,19.584,152.812
C07107=1092.604,229.623,-74.427,176.864,19.586,152.812
C07108=1092.609,229.872,-74.453,176.867,19.588,152.812
C07109=1092.616,230.121,-74.479,176.870,19.590,152.812
C07110=1092.620,230.369,-74.504,176.873,19.592,152.811
C07111=1092.627,230.618,-74.530,176.876,19.594,152.811
C07112=1092.632,230.867,-74.556,176.879,19.596,152.811
C07113=1092.638,231.115,-74.582,176.882,19.598,152.811
C07114=1092.643,231.363,-74.607,176.884,19.600,152.811
C07115=1092.649,231.612,-74.633,176.888,19.602,152.811
C07116=1092.654,231.861,-74.659,176.891,19.604,152.811
C07117=1092.660,232.110,-74.685,176.894,19.605,152.811
C07118=1092.665,232.358,-74.710,176.897,19.607,152.811
C07119=1092.671,232.606,-74.737,176.900,19.609,152.811
C07120=1092.677,232.855,-74.762,176.903,19.611,152.810
C07121=1092.683,233.104,-74.788,176.906,19.613,152.810
C07122=1092.688,233.352,-74.813,176.909,19.615,152.810
C07123=1092.693,233.601,-74.839,176.912,19.617,152.810
C07124=1092.699,233.850,-74.866,176.915,19.618,152.810
C07125=1092.705,234.099,-74.892,176.918,19.621,152.810
C07126=1092.711,234.347,-74.917,176.920,19.623,152.810
C07127=1092.716,234.596,-74.944,176.924,19.625,152.810
C07128=1092.721,234.844,-74.969,176.927,19.627,152.810
C07129=1092.727,235.093,-74.995,176.929,19.628,152.810
C07130=1092.732,235.342,-75.021,176.933,19.631,152.810
C07131=1092.741,235.715,-75.061,176.937,19.633,152.809
C07132=1092.750,236.088,-75.099,176.942,19.637,152.809
C07133=1092.758,236.461,-75.139,176.946,19.639,152.809
C07134=1092.766,236.833,-75.178,176.951,19.643,152.809
C07135=1092.772,237.082,-75.204,176.954,19.644,152.809
C07136=1092.777,237.331,-75.230,176.957,19.646,152.809
C07137=1092.783,237.579,-75.257,176.959,19.648,152.809
C07138=1092.788,237.828,-75.283,176.963,19.650,152.809
C07139=1092.795,238.076,-75.309,176.966,19.652,152.808
C07140=1092.800,238.325,-75.335,176.969,19.654,152.808
C07141=1092.806,238.574,-75.361,176.972,19.656,152.808
C07142=1092.812,238.823,-75.387,176.974,19.658,152.808
C07143=1092.817,239.070,-75.413,176.978,19.660,152.808
C07144=1092.822,239.319,-75.439,176.981,19.662,152.808
C07145=1092.828,239.567,-75.466,176.984,19.664,152.808
C07146=1092.834,239.816,-75.493,176.987,19.666,152.808
C07147=1092.839,240.065,-75.519,176.990,19.668,152.808
C07148=1092.845,240.313,-75.545,176.993,19.669,152.808
C07149=1092.850,240.562,-75.571,176.996,19.671,152.808
C07150=1092.856,240.811,-75.598,177.000,19.674,152.807
C07151=1092.862,241.059,-75.624,177.002,19.675,152.807
C07152=1092.867,241.308,-75.650,177.005,19.678,152.807
C07153=1092.873,241.556,-75.677,177.008,19.679,152.807
C07154=1092.879,241.805,-75.704,177.011,19.681,152.807
C07155=1092.884,242.054,-75.730,177.014,19.684,152.807
C07156=1092.890,242.302,-75.756,177.017,19.685,152.807
C07157=1092.896,242.550,-75.783,177.020,19.687,152.807
C07158=1092.901,242.799,-75.809,177.024,19.689,152.807
C07159=1092.907,243.048,-75.835,177.026,19.691,152.807
C07160=1092.913,243.296,-75.862,177.030,19.693,152.807
C07161=1092.919,243.544,-75.889,177.033,19.696,152.807
C07162=1092.924,243.794,-75.915,177.035,19.697,152.806
C07163=1092.929,244.042,-75.942,177.039,19.699,152.806
C07164=1092.935,244.290,-75.969,177.042,19.701,152.806
C07165=1092.941,244.539,-75.995,177.044,19.703,152.806
C07166=1092.947,244.787,-76.022,177.048,19.706,152.806
C07167=1092.952,245.036,-76.048,177.051,19.708,152.806
C07168=1092.957,245.285,-76.075,177.053,19.709,152.806
C07169=1092.963,245.533,-76.102,177.057,19.711,152.806
C07170=1092.969,245.781,-76.128,177.060,19.713,152.806
C07171=1092.974,246.030,-76.155,177.062,19.716,152.806
C07172=1092.980,246.278,-76.182,177.066,19.718,152.806
C07173=1092.985,246.527,-76.209,177.069,19.720,152.806
C07174=1092.991,246.775,-76.236,177.072,19.721,152.806
C07175=1092.997,247.024,-76.262,177.075,19.723,152.805
C07176=1093.002,247.272,-76.289,177.078,19.726,152.805
C07177=1093.008,247.521,-76.316,177.081,19.728,152.805
C07178=1093.014,247.770,-76.343,177.084,19.730,152.805
C07179=1093.019,248.018,-76.370,177.087,19.732,152.805
C07180=1093.025,248.267,-76.397,177.090,19.734,152.805
C07181=1093.031,248.515,-76.424,177.093,19.736,152.805
C07182=1093.036,248.764,-76.451,177.096,19.738,152.805
C07183=1093.044,249.130,-76.490,177.100,19.741,152.805
C07184=1093.052,249.496,-76.530,177.105,19.744,152.805
C07185=1093.060,249.862,-76.569,177.110,19.747,152.805
C07186=1093.068,250.228,-76.610,177.114,19.751,152.805
C07187=1093.074,250.476,-76.637,177.117,19.752,152.805
C07188=1093.079,250.725,-76.664,177.120,19.754,152.804
C07189=1093.085,250.973,-76.691,177.123,19.757,152.804
C07190=1093.090,251.222,-76.717,177.126,19.758,152.804
C07191=1093.095,251.470,-76.744,177.129,19.761,152.804
C07192=1093.101,251.719,-76.771,177.132,19.763,152.804
C07193=1093.107,251.968,-76.799,177.136,19.765,152.804
C07194=1093.113,252.216,-76.826,177.138,19.767,152.804
C07195=1093.118,252.465,-76.853,177.142,19.769,152.804
C07196=1093.124,252.713,-76.880,177.145,19.771,152.804
C07197=1093.129,252.961,-76.908,177.147,19.773,152.804
C07198=1093.135,253.209,-76.935,177.151,19.775,152.804
C07199=1093.141,253.459,-76.962,177.154,19.778,152.804
C07200=1093.147,253.706,-76.990,177.157,19.780,152.804
C07201=1093.152,253.955,-77.017,177.160,19.781,152.804
C07202=1093.157,254.203,-77.043,177.163,19.783,152.804
C07203=1093.163,254.452,-77.071,177.166,19.786,152.804
C07204=1093.169,254.701,-77.098,177.169,19.788,152.803
C07205=1093.174,254.949,-77.126,177.172,19.790,152.803
C07206=1093.180,255.197,-77.154,177.175,19.792,152.803
C07207=1093.185,255.446,-77.180,177.179,19.794,152.803
C07208=1093.191,255.695,-77.208,177.181,19.796,152.803
C07209=1093.197,255.943,-77.235,177.184,19.798,152.803
C07210=1093.202,256.191,-77.262,177.188,19.801,152.803
C07211=1093.208,256.439,-77.290,177.191,19.803,152.803
C07212=1093.214,256.689,-77.317,177.193,19.804,152.803
C07213=1093.219,256.937,-77.345,177.197,19.806,152.803
C07214=1093.225,257.185,-77.372,177.200,19.809,152.803
C07215=1093.230,257.433,-77.400,177.203,19.811,152.803
C07216=1093.237,257.682,-77.427,177.206,19.813,152.803
C07217=1093.242,257.930,-77.455,177.209,19.815,152.803
C07218=1093.247,258.179,-77.482,177.212,19.817,152.803
C07219=1093.254,258.427,-77.510,177.216,19.820,152.802
C07220=1093.259,258.676,-77.537,177.218,19.821,152.802
C07221=1093.265,258.924,-77.565,177.221,19.824,152.802
C07222=1093.271,259.172,-77.593,177.225,19.826,152.802
C07223=1093.276,259.421,-77.620,177.228,19.828,152.802
C07224=1093.282,259.669,-77.647,177.231,19.829,152.802
C07225=1093.288,259.918,-77.676,177.234,19.832,152.802
C07226=1093.293,260.166,-77.703,177.237,19.834,152.802
C07227=1093.299,260.414,-77.730,177.240,19.836,152.802
C07228=1093.305,260.663,-77.759,177.243,19.838,152.802
C07229=1093.310,260.911,-77.786,177.246,19.840,152.802
C07230=1093.317,261.160,-77.814,177.249,19.843,152.802
C07231=1093.322,261.408,-77.842,177.253,19.845,152.802
C07232=1093.327,261.657,-77.869,177.255,19.847,152.802
C07233=1093.334,261.905,-77.897,177.258,19.849,152.802
C07234=1093.339,262.153,-77.925,177.262,19.851,152.802
C07235=1093.347,262.517,-77.966,177.266,19.854,152.801
C07236=1093.356,262.879,-78.006,177.271,19.857,152.801
C07237=1093.364,263.243,-78.047,177.276,19.860,152.801
C07238=1093.372,263.606,-78.087,177.280,19.863,152.801
C07239=1093.379,263.855,-78.115,177.283,19.865,152.801
C07240=1093.384,264.103,-78.143,177.287,19.868,152.801
C07241=1093.390,264.351,-78.171,177.289,19.869,152.801
C07242=1093.396,264.599,-78.199,177.292,19.872,152.801
C07243=1093.401,264.848,-78.227,177.296,19.874,152.801
C07244=1093.407,265.096,-78.256,177.299,19.876,152.801
C07245=1093.413,265.345,-78.282,177.302,19.879,152.801
C07246=1093.419,265.593,-78.311,177.304,19.881,152.801
C07247=1093.424,265.841,-78.339,177.308,19.883,152.801
C07248=1093.429,266.089,-78.367,177.311,19.885,152.801
C07249=1093.435,266.338,-78.395,177.314,19.887,152.801
C07250=1093.441,266.586,-78.423,177.318,19.889,152.801
C07251=1093.447,266.835,-78.451,177.320,19.892,152.801
C07252=1093.452,267.083,-78.479,177.323,19.894,152.801
C07253=1093.458,267.332,-78.508,177.326,19.896,152.801
C07254=1093.464,267.579,-78.536,177.330,19.898,152.801
C07255=1093.469,267.828,-78.565,177.333,19.901,152.801
C07256=1093.475,268.076,-78.592,177.335,19.902,152.800
C07257=1093.481,268.325,-78.621,177.339,19.905,152.800
C07258=1093.486,268.573,-78.649,177.342,19.907,152.800
C07259=1093.492,268.822,-78.677,177.345,19.909,152.800
C07260=1093.497,269.070,-78.705,177.348,19.912,152.800
C07261=1093.503,269.318,-78.733,177.352,19.914,152.800
C07262=1093.509,269.566,-78.762,177.354,19.916,152.800
C07263=1093.514,269.815,-78.791,177.357,19.918,152.800
C07264=1093.520,270.063,-78.819,177.360,19.921,152.800
C07265=1093.525,270.312,-78.847,177.364,19.923,152.800
C07266=1093.531,270.560,-78.875,177.367,19.925,152.800
C07267=1093.537,270.808,-78.904,177.370,19.927,152.800
C07268=1093.542,271.056,-78.932,177.373,19.929,152.800
C07269=1093.548,271.305,-78.961,177.376,19.932,152.800
C07270=1093.554,271.553,-78.988,177.379,19.934,152.800
C07271=1093.559,271.801,-79.018,177.382,19.936,152.800
C07272=1093.565,272.050,-79.046,177.386,19.939,152.800
C07273=1093.570,272.298,-79.074,177.389,19.941,152.800
C07274=1093.577,272.546,-79.103,177.391,19.943,152.800
C07275=1093.582,272.794,-79.131,177.395,19.945,152.800
C07276=1093.587,273.043,-79.160,177.398,19.948,152.800
C07277=1093.593,273.291,-79.189,177.401,19.950,152.800
C07278=1093.599,273.539,-79.217,177.404,19.952,152.800
C07279=1093.605,273.788,-79.246,177.407,19.955,152.800
C07280=1093.610,274.036,-79.274,177.411,19.957,152.800
C07281=1093.616,274.285,-79.303,177.413,19.959,152.800
C07282=1093.621,274.532,-79.332,177.416,19.961,152.800
C07283=1093.627,274.781,-79.360,177.420,19.964,152.800
C07284=1093.633,275.029,-79.390,177.423,19.966,152.800
